C07312=1171.971,266.209,-67.189,-177.179,7.557,148.617
C07313=1171.975,265.960,-67.160,-177.181,7.554,148.617
C07314=1171.979,265.712,-67.133,-177.184,7.552,148.617
C07315=1171.984,265.463,-67.104,-177.186,7.549,148.617
C07316=1171.988,265.215,-67.077,-177.189,7.546,148.617
C07317=1171.992,264.966,-67.049,-177.192,7.543,148.617
C07318=1171.997,264.718,-67.020,-177.194,7.541,148.617
C07319=1172.002,264.470,-66.993,-177.197,7.538,148.617
C07320=1172.005,264.222,-66.964,-177.200,7.535,148.618
C07321=1172.011,263.973,-66.937,-177.202,7.532,148.618
C07322=1172.014,263.724,-66.909,-177.205,7.530,148.618
C07323=1172.019,263.476,-66.881,-177.208,7.527,148.618
C07324=1172.023,263.228,-66.853,-177.210,7.524,148.618
C07325=1172.028,262.979,-66.825,-177.213,7.521,148.618
C07326=1172.032,262.731,-66.797,-177.215,7.519,148.618
C07327=1172.037,262.458,-66.767,-177.219,7.515,148.618
C07328=1172.042,262.184,-66.736,-177.221,7.512,148.618
C07329=1172.047,261.912,-66.706,-177.224,7.509,148.618
C07330=1172.052,261.638,-66.675,-177.227,7.507,148.619
C07331=1172.055,261.390,-66.647,-177.230,7.504,148.619
C07332=1172.060,261.142,-66.619,-177.232,7.502,148.619
C07333=1172.064,260.894,-66.592,-177.235,7.499,148.619
C07334=1172.068,260.645,-66.564,-177.238,7.496,148.619
C07335=1172.073,260.396,-66.536,-177.241,7.493,148.619
C07336=1172.078,260.148,-66.508,-177.243,7.491,148.619
C07337=1172.082,259.900,-66.480,-177.245,7.488,148.619
C07338=1172.086,259.651,-66.453,-177.248,7.485,148.619
C07339=1172.091,259.403,-66.425,-177.251,7.482,148.619
C07340=1172.095,259.154,-66.398,-177.254,7.480,148.619
C07341=1172.099,258.906,-66.370,-177.256,7.477,148.619
C07342=1172.104,258.658,-66.343,-177.259,7.474,148.620
C07343=1172.107,258.409,-66.315,-177.261,7.472,148.620
C07344=1172.113,258.160,-66.287,-177.264,7.469,148.620
C07345=1172.117,257.913,-66.260,-177.267,7.466,148.620
C07346=1172.121,257.663,-66.232,-177.270,7.463,148.620
C07347=1172.126,257.415,-66.204,-177.272,7.461,148.620
C07348=1172.130,257.167,-66.177,-177.275,7.458,148.620
C07349=1172.135,256.919,-66.149,-177.278,7.455,148.620
C07350=1172.139,256.670,-66.122,-177.280,7.453,148.620
C07351=1172.143,256.421,-66.095,-177.283,7.450,148.620
C07352=1172.148,256.173,-66.067,-177.285,7.447,148.620
C07353=1172.152,255.924,-66.040,-177.288,7.444,148.620
C07354=1172.156,255.676,-66.013,-177.290,7.442,148.621
C07355=1172.161,255.428,-65.985,-177.294,7.439,148.621
C07356=1172.165,255.179,-65.958,-177.296,7.436,148.621
C07357=1172.170,254.931,-65.931,-177.298,7.434,148.621
C07358=1172.174,254.682,-65.903,-177.301,7.431,148.621
C07359=1172.178,254.434,-65.876,-177.304,7.428,148.621
C07360=1172.183,254.185,-65.849,-177.306,7.426,148.621
C07361=1172.187,253.937,-65.821,-177.309,7.424,148.622
C07362=1172.191,253.688,-65.793,-177.312,7.421,148.622
C07363=1172.196,253.440,-65.766,-177.315,7.418,148.622
C07364=1172.200,253.192,-65.740,-177.317,7.415,148.622
C07365=1172.204,252.944,-65.712,-177.320,7.413,148.622
C07366=1172.209,252.695,-65.685,-177.323,7.410,148.622
C07367=1172.213,252.446,-65.658,-177.325,7.408,148.622
C07368=1172.218,252.198,-65.631,-177.328,7.405,148.622
C07369=1172.222,251.949,-65.603,-177.331,7.402,148.622
C07370=1172.227,251.701,-65.576,-177.333,7.400,148.622
C07371=1172.231,251.453,-65.549,-177.336,7.397,148.622
C07372=1172.235,251.204,-65.522,-177.339,7.394,148.623
C07373=1172.239,250.955,-65.495,-177.341,7.392,148.623
C07374=1172.244,250.707,-65.468,-177.344,7.389,148.623
C07375=1172.249,250.458,-65.441,-177.346,7.386,148.623
C07376=1172.253,250.210,-65.414,-177.349,7.384,148.623
C07377=1172.258,249.961,-65.386,-177.352,7.381,148.623
C07378=1172.262,249.713,-65.360,-177.355,7.378,148.623
C07379=1172.266,249.464,-65.333,-177.357,7.376,148.623
C07380=1172.271,249.215,-65.306,-177.360,7.373,148.624
C07381=1172.275,248.967,-65.278,-177.363,7.371,148.624
C07382=1172.280,248.718,-65.251,-177.365,7.368,148.624
C07383=1172.284,248.470,-65.225,-177.368,7.365,148.624
C07384=1172.289,248.222,-65.198,-177.370,7.362,148.624
C07385=1172.293,247.973,-65.171,-177.373,7.360,148.624
C07386=1172.298,247.725,-65.144,-177.376,7.358,148.624
C07387=1172.302,247.477,-65.117,-177.379,7.355,148.624
C07388=1172.306,247.228,-65.090,-177.381,7.353,148.625
C07389=1172.310,246.979,-65.063,-177.384,7.350,148.625
C07390=1172.314,246.731,-65.036,-177.386,7.348,148.625
C07391=1172.319,246.482,-65.009,-177.389,7.345,148.625
C07392=1172.324,246.234,-64.982,-177.392,7.342,148.625
C07393=1172.328,245.985,-64.956,-177.394,7.340,148.625
C07394=1172.333,245.736,-64.929,-177.397,7.337,148.625
C07395=1172.337,245.488,-64.902,-177.400,7.334,148.626
C07396=1172.341,245.240,-64.876,-177.402,7.332,148.626
C07397=1172.346,244.991,-64.849,-177.405,7.329,148.626
C07398=1172.350,244.743,-64.822,-177.408,7.326,148.626
C07399=1172.355,244.494,-64.796,-177.410,7.324,148.626
C07400=1172.359,244.245,-64.769,-177.413,7.321,148.626
C07401=1172.364,243.997,-64.742,-177.416,7.320,148.627
C07402=1172.368,243.749,-64.715,-177.418,7.317,148.627
C07403=1172.373,243.500,-64.689,-177.421,7.314,148.627
C07404=1172.377,243.251,-64.663,-177.423,7.311,148.627
C07405=1172.381,243.003,-64.636,-177.427,7.309,148.627
C07406=1172.386,242.754,-64.610,-177.429,7.306,148.627
C07407=1172.390,242.506,-64.583,-177.431,7.304,148.627
C07408=1172.395,242.257,-64.556,-177.435,7.301,148.627
C07409=1172.399,242.008,-64.530,-177.437,7.299,148.628
C07410=1172.404,241.760,-64.503,-177.440,7.296,148.628
C07411=1172.408,241.512,-64.476,-177.443,7.293,148.628
C07412=1172.413,241.263,-64.450,-177.445,7.291,148.628
C07413=1172.417,241.014,-64.424,-177.448,7.288,148.628
C07414=1172.421,240.766,-64.396,-177.450,7.287,148.628
C07415=1172.426,240.517,-64.371,-177.453,7.284,148.629
C07416=1172.430,240.269,-64.344,-177.456,7.281,148.629
C07417=1172.434,240.020,-64.318,-177.458,7.278,148.629
C07418=1172.439,239.771,-64.291,-177.461,7.276,148.629
C07419=1172.443,239.522,-64.265,-177.464,7.274,148.629
C07420=1172.448,239.274,-64.238,-177.466,7.271,148.629
C07421=1172.453,239.026,-64.213,-177.469,7.268,148.629
C07422=1172.457,238.778,-64.186,-177.472,7.266,148.630
C07423=1172.462,238.529,-64.160,-177.474,7.263,148.630
C07424=1172.466,238.280,-64.133,-177.477,7.261,148.630
C07425=1172.471,238.031,-64.107,-177.480,7.258,148.630
C07426=1172.475,237.783,-64.081,-177.482,7.256,148.630
C07427=1172.479,237.534,-64.054,-177.485,7.253,148.630
C07428=1172.483,237.286,-64.028,-177.488,7.251,148.630
C07429=1172.488,237.037,-64.002,-177.491,7.249,148.631
C07430=1172.493,236.789,-63.976,-177.493,7.246,148.631
C07431=1172.498,236.517,-63.947,-177.496,7.243,148.631
C07432=1172.502,236.245,-63.919,-177.499,7.240,148.631
C07433=1172.507,235.974,-63.890,-177.502,7.238,148.631
C07434=1172.512,235.702,-63.862,-177.505,7.235,148.632
C07435=1172.516,235.454,-63.835,-177.508,7.232,148.632
C07436=1172.521,235.205,-63.809,-177.510,7.231,148.632
C07437=1172.525,234.956,-63.783,-177.513,7.228,148.632
C07438=1172.530,234.708,-63.757,-177.516,7.225,148.632
C07439=1172.535,234.459,-63.731,-177.518,7.223,148.632
C07440=1172.539,234.210,-63.705,-177.521,7.220,148.633
C07441=1172.543,233.962,-63.679,-177.524,7.218,148.633
C07442=1172.548,233.713,-63.652,-177.527,7.215,148.633
C07443=1172.553,233.465,-63.627,-177.529,7.213,148.633
C07444=1172.557,233.216,-63.601,-177.532,7.210,148.633
C07445=1172.561,232.967,-63.575,-177.534,7.208,148.633
C07446=1172.566,232.719,-63.548,-177.537,7.206,148.634
C07447=1172.570,232.470,-63.523,-177.540,7.204,148.634
C07448=1172.575,232.222,-63.497,-177.542,7.201,148.634
C07449=1172.579,231.973,-63.471,-177.546,7.198,148.634
C07450=1172.583,231.724,-63.446,-177.548,7.196,148.634
C07451=1172.588,231.475,-63.419,-177.551,7.193,148.635
C07452=1172.593,231.228,-63.393,-177.553,7.191,148.635
C07453=1172.597,230.979,-63.367,-177.556,7.188,148.635
C07454=1172.601,230.730,-63.342,-177.559,7.186,148.635
C07455=1172.605,230.481,-63.316,-177.561,7.183,148.635
C07456=1172.610,230.233,-63.291,-177.564,7.182,148.636
C07457=1172.615,229.984,-63.264,-177.567,7.179,148.636
C07458=1172.619,229.735,-63.239,-177.569,7.177,148.636
C07459=1172.624,229.487,-63.213,-177.572,7.174,148.636
C07460=1172.628,229.238,-63.187,-177.574,7.172,148.636
C07461=1172.633,228.990,-63.162,-177.578,7.169,148.636
C07462=1172.637,228.741,-63.136,-177.580,7.167,148.637
C07463=1172.642,228.493,-63.110,-177.583,7.164,148.637
C07464=1172.646,228.244,-63.085,-177.585,7.162,148.637
C07465=1172.650,227.995,-63.059,-177.588,7.160,148.637
C07466=1172.655,227.746,-63.033,-177.591,7.157,148.637
C07467=1172.660,227.498,-63.007,-177.594,7.155,148.638
C07468=1172.664,227.249,-62.982,-177.596,7.153,148.638
C07469=1172.668,227.000,-62.956,-177.599,7.150,148.638
C07470=1172.673,226.752,-62.930,-177.601,7.148,148.638
C07471=1172.678,226.503,-62.905,-177.604,7.145,148.638
C07472=1172.682,226.254,-62.880,-177.607,7.143,148.639
C07473=1172.687,226.006,-62.854,-177.610,7.140,148.639
C07474=1172.691,225.757,-62.828,-177.612,7.138,148.639
C07475=1172.696,225.509,-62.803,-177.615,7.136,148.639
C07476=1172.700,225.260,-62.777,-177.618,7.134,148.639
C07477=1172.704,225.011,-62.752,-177.620,7.131,148.640
C07478=1172.709,224.763,-62.727,-177.623,7.129,148.640
C07479=1172.714,224.514,-62.701,-177.626,7.126,148.640
C07480=1172.718,224.265,-62.675,-177.628,7.124,148.640
C07481=1172.723,224.017,-62.650,-177.631,7.121,148.640
C07482=1172.727,223.767,-62.625,-177.634,7.119,148.641
C07483=1172.732,223.519,-62.600,-177.637,7.117,148.641
C07484=1172.736,223.271,-62.574,-177.639,7.115,148.641
C07485=1172.740,223.022,-62.549,-177.642,7.112,148.641
C07486=1172.745,222.773,-62.524,-177.645,7.110,148.642
C07487=1172.749,222.525,-62.498,-177.647,7.108,148.642
C07488=1172.754,222.276,-62.473,-177.650,7.105,148.642
C07489=1172.758,222.027,-62.448,-177.652,7.103,148.642
C07490=1172.763,221.779,-62.422,-177.656,7.100,148.642
C07491=1172.768,221.530,-62.397,-177.658,7.098,148.642
C07492=1172.772,221.281,-62.372,-177.661,7.096,148.643
C07493=1172.777,221.033,-62.346,-177.663,7.094,148.643
C07494=1172.781,220.783,-62.322,-177.666,7.091,148.643
C07495=1172.786,220.535,-62.296,-177.669,7.089,148.643
C07496=1172.790,220.287,-62.271,-177.672,7.086,148.644
C07497=1172.795,220.038,-62.246,-177.674,7.084,148.644
C07498=1172.799,219.789,-62.220,-177.677,7.082,148.644
C07499=1172.803,219.541,-62.196,-177.679,7.079,148.644
C07500=1172.808,219.292,-62.170,-177.682,7.078,148.644
C07501=1172.813,219.043,-62.146,-177.685,7.075,148.645
C07502=1172.817,218.794,-62.120,-177.688,7.073,148.645
C07503=1172.822,218.546,-62.095,-177.690,7.070,148.645
C07504=1172.826,218.297,-62.070,-177.693,7.068,148.645
C07505=1172.831,218.048,-62.046,-177.696,7.065,148.646
C07506=1172.835,217.800,-62.020,-177.698,7.063,148.646
C07507=1172.840,217.551,-61.995,-177.701,7.062,148.646
C07508=1172.844,217.302,-61.970,-177.704,7.059,148.646
C07509=1172.849,217.054,-61.945,-177.706,7.057,148.646
C07510=1172.853,216.804,-61.920,-177.709,7.054,148.647
C07511=1172.857,216.556,-61.895,-177.712,7.052,148.647
C07512=1172.862,216.307,-61.870,-177.714,7.050,148.647
C07513=1172.867,216.059,-61.845,-177.717,7.047,148.647
C07514=1172.871,215.809,-61.820,-177.720,7.046,148.648
C07515=1172.876,215.561,-61.796,-177.723,7.043,148.648
C07516=1172.880,215.312,-61.770,-177.725,7.041,148.648
C07517=1172.885,215.063,-61.746,-177.728,7.038,148.648
C07518=1172.889,214.815,-61.721,-177.731,7.036,148.649
C07519=1172.894,214.566,-61.696,-177.733,7.034,148.649
C07520=1172.898,214.318,-61.672,-177.736,7.031,148.649
C07521=1172.903,214.068,-61.647,-177.739,7.030,148.649
C07522=1172.908,213.820,-61.622,-177.742,7.027,148.649
C07523=1172.911,213.571,-61.597,-177.744,7.025,148.650
C07524=1172.916,213.322,-61.572,-177.747,7.023,148.650
C07525=1172.921,213.074,-61.547,-177.750,7.020,148.650
C07526=1172.925,212.825,-61.523,-177.752,7.018,148.650
C07527=1172.930,212.577,-61.498,-177.755,7.015,148.651
C07528=1172.934,212.328,-61.474,-177.758,7.014,148.651
C07529=1172.939,212.079,-61.448,-177.760,7.011,148.651
C07530=1172.943,211.830,-61.424,-177.763,7.009,148.651
C07531=1172.948,211.581,-61.399,-177.765,7.007,148.651
C07532=1172.953,211.332,-61.375,-177.768,7.005,148.652
C07533=1172.957,211.084,-61.350,-177.771,7.002,148.652
C07534=1172.962,210.835,-61.325,-177.774,7.000,148.652
C07535=1172.967,210.565,-61.298,-177.777,6.998,148.653
C07536=1172.972,210.294,-61.273,-177.780,6.995,148.653
C07537=1172.976,210.023,-61.246,-177.782,6.993,148.653
C07538=1172.981,209.753,-61.219,-177.785,6.990,148.653
C07539=1172.986,209.505,-61.194,-177.788,6.988,148.654
C07540=1172.990,209.255,-61.170,-177.791,6.985,148.654
C07541=1172.995,209.007,-61.145,-177.794,6.984,148.654
C07542=1173.000,208.758,-61.121,-177.796,6.982,148.654
C07543=1173.005,208.510,-61.096,-177.799,6.979,148.655
C07544=1173.009,208.260,-61.072,-177.802,6.977,148.655
C07545=1173.014,208.012,-61.047,-177.804,6.975,148.655
C07546=1173.018,207.763,-61.023,-177.807,6.972,148.655
C07547=1173.022,207.514,-60.999,-177.810,6.971,148.656
C07548=1173.027,207.265,-60.974,-177.813,6.968,148.656
C07549=1173.031,207.017,-60.950,-177.815,6.966,148.656
C07550=1173.037,206.768,-60.925,-177.818,6.964,148.656
C07551=1173.040,206.519,-60.901,-177.821,6.961,148.657
C07552=1173.045,206.271,-60.877,-177.823,6.959,148.657
C07553=1173.050,206.022,-60.852,-177.826,6.958,148.657
C07554=1173.054,205.774,-60.828,-177.829,6.955,148.657
C07555=1173.059,205.524,-60.804,-177.831,6.953,148.658
C07556=1173.064,205.275,-60.780,-177.834,6.951,148.658
C07557=1173.068,205.027,-60.756,-177.837,6.948,148.658
C07558=1173.073,204.778,-60.731,-177.839,6.946,148.658
C07559=1173.077,204.529,-60.707,-177.842,6.945,148.659
C07560=1173.081,204.281,-60.683,-177.845,6.942,148.659
C07561=1173.087,204.031,-60.659,-177.848,6.940,148.659
C07562=1173.091,203.783,-60.634,-177.850,6.938,148.659
C07563=1173.096,203.534,-60.610,-177.853,6.935,148.660
C07564=1173.099,203.285,-60.586,-177.856,6.933,148.660
C07565=1173.105,203.036,-60.562,-177.858,6.931,148.660
C07566=1173.109,202.788,-60.538,-177.861,6.929,148.660
C07567=1173.114,202.539,-60.514,-177.864,6.927,148.661
C07568=1173.118,202.291,-60.490,-177.866,6.925,148.661
C07569=1173.123,202.041,-60.465,-177.869,6.922,148.661
C07570=1173.127,201.792,-60.441,-177.872,6.920,148.662
C07571=1173.132,201.544,-60.417,-177.875,6.918,148.662
C07572=1173.136,201.295,-60.394,-177.877,6.916,148.662
C07573=1173.141,201.046,-60.369,-177.880,6.914,148.662
C07574=1173.146,200.798,-60.345,-177.883,6.912,148.663
C07575=1173.150,200.548,-60.321,-177.885,6.910,148.663
C07576=1173.154,200.299,-60.297,-177.888,6.907,148.663
C07577=1173.159,200.050,-60.274,-177.891,6.905,148.664
C07578=1173.164,199.802,-60.249,-177.893,6.903,148.664
C07579=1173.168,199.553,-60.225,-177.896,6.901,148.664
C07580=1173.173,199.304,-60.202,-177.899,6.899,148.664
C07581=1173.178,199.056,-60.178,-177.901,6.897,148.664
C07582=1173.182,198.807,-60.155,-177.904,6.894,148.665
C07583=1173.187,198.558,-60.130,-177.907,6.892,148.665
C07584=1173.191,198.309,-60.107,-177.910,6.891,148.665
C07585=1173.196,198.060,-60.082,-177.912,6.889,148.666
C07586=1173.201,197.811,-60.059,-177.915,6.886,148.666
C07587=1173.205,197.563,-60.035,-177.918,6.884,148.666
C07588=1173.210,197.313,-60.011,-177.920,6.882,148.666
C07589=1173.214,197.065,-59.987,-177.923,6.879,148.667
C07590=1173.219,196.816,-59.964,-177.926,6.878,148.667
C07591=1173.223,196.568,-59.940,-177.929,6.876,148.667
C07592=1173.228,196.319,-59.916,-177.931,6.874,148.668
C07593=1173.233,196.070,-59.893,-177.934,6.871,148.668
C07594=1173.237,195.821,-59.869,-177.937,6.869,148.668
C07595=1173.242,195.572,-59.846,-177.939,6.867,148.668
C07596=1173.246,195.324,-59.822,-177.942,6.865,148.669
C07597=1173.251,195.075,-59.798,-177.945,6.863,148.669
C07598=1173.255,194.826,-59.775,-177.947,6.861,148.669
C07599=1173.260,194.577,-59.751,-177.950,6.859,148.670
C07600=1173.264,194.328,-59.727,-177.953,6.856,148.670
C07601=1173.269,194.078,-59.704,-177.956,6.855,148.670
C07602=1173.273,193.830,-59.680,-177.958,6.853,148.671
C07603=1173.278,193.581,-59.656,-177.960,6.851,148.671
C07604=1173.282,193.332,-59.633,-177.964,6.848,148.671
C07605=1173.287,193.083,-59.610,-177.966,6.846,148.671
C07606=1173.292,192.835,-59.585,-177.969,6.845,148.672
C07607=1173.297,192.586,-59.562,-177.971,6.842,148.672
C07608=1173.302,192.337,-59.539,-177.974,6.840,148.672
C07609=1173.306,192.088,-59.516,-177.977,6.838,148.673
C07610=1173.311,191.840,-59.492,-177.980,6.836,148.673
C07611=1173.315,191.591,-59.468,-177.982,6.834,148.673
C07612=1173.320,191.342,-59.445,-177.985,6.832,148.673
C07613=1173.325,191.093,-59.422,-177.988,6.830,148.674
C07614=1173.329,190.844,-59.398,-177.991,6.828,148.674
C07615=1173.334,190.595,-59.374,-177.993,6.826,148.674
C07616=1173.338,190.346,-59.351,-177.996,6.824,148.675
C07617=1173.343,190.097,-59.328,-177.999,6.822,148.675
C07618=1173.347,189.848,-59.305,-178.001,6.820,148.675
C07619=1173.352,189.599,-59.281,-178.004,6.818,148.675
C07620=1173.357,189.350,-59.258,-178.006,6.816,148.676
C07621=1173.361,189.101,-59.235,-178.010,6.813,148.676
C07622=1173.366,188.852,-59.211,-178.012,6.811,148.676
C07623=1173.370,188.604,-59.188,-178.014,6.809,148.677
C07624=1173.375,188.355,-59.165,-178.017,6.808,148.677
C07625=1173.380,188.106,-59.142,-178.020,6.805,148.677
C07626=1173.385,187.857,-59.119,-178.023,6.803,148.678
C07627=1173.389,187.608,-59.095,-178.026,6.801,148.678
C07628=1173.393,187.359,-59.073,-178.028,6.799,148.678
C07629=1173.398,187.110,-59.049,-178.031,6.798,148.678
C07630=1173.403,186.861,-59.026,-178.034,6.795,148.679
C07631=1173.407,186.612,-59.003,-178.037,6.793,148.679
C07632=1173.412,186.364,-58.980,-178.039,6.791,148.679
C07633=1173.417,186.115,-58.957,-178.041,6.789,148.680
C07634=1173.421,185.866,-58.933,-178.044,6.787,148.680
C07635=1173.426,185.617,-58.910,-178.047,6.785,148.680
C07636=1173.430,185.368,-58.887,-178.050,6.783,148.681
C07637=1173.435,185.119,-58.864,-178.053,6.781,148.681
C07638=1173.439,184.870,-58.841,-178.055,6.779,148.681
C07639=1173.444,184.601,-58.816,-178.058,6.777,148.681
C07640=1173.449,184.331,-58.791,-178.061,6.775,148.682
C07641=1173.455,184.061,-58.766,-178.064,6.772,148.682
C07642=1173.459,183.792,-58.742,-178.067,6.771,148.682
C07643=1173.465,183.544,-58.719,-178.069,6.769,148.683
C07644=1173.469,183.295,-58.695,-178.072,6.767,148.683
C07645=1173.473,183.046,-58.673,-178.075,6.764,148.684
C07646=1173.478,182.797,-58.649,-178.078,6.763,148.684
C07647=1173.483,182.547,-58.627,-178.080,6.760,148.684
C07648=1173.487,182.299,-58.604,-178.083,6.759,148.684
C07649=1173.492,182.050,-58.581,-178.086,6.757,148.685
C07650=1173.496,181.801,-58.558,-178.088,6.755,148.685
C07651=1173.501,181.552,-58.535,-178.091,6.753,148.685
C07652=1173.506,181.303,-58.512,-178.094,6.751,148.686
C07653=1173.510,181.055,-58.490,-178.096,6.749,148.686
C07654=1173.515,180.806,-58.466,-178.099,6.747,148.686
C07655=1173.519,180.556,-58.444,-178.102,6.745,148.687
C07656=1173.524,180.307,-58.421,-178.104,6.743,148.687
C07657=1173.529,180.059,-58.398,-178.108,6.741,148.687
C07658=1173.534,179.810,-58.376,-178.110,6.739,148.688
C07659=1173.538,179.561,-58.352,-178.113,6.737,148.688
C07660=1173.542,179.312,-58.330,-178.115,6.735,148.688
C07661=1173.548,179.063,-58.307,-178.118,6.733,148.689
C07662=1173.552,178.814,-58.285,-178.121,6.732,148.689
C07663=1173.557,178.565,-58.262,-178.124,6.729,148.689
C07664=1173.561,178.317,-58.240,-178.127,6.727,148.690
C07665=1173.566,178.068,-58.216,-178.129,6.725,148.690
C07666=1173.570,177.818,-58.194,-178.131,6.723,148.690
C07667=1173.576,177.570,-58.171,-178.134,6.722,148.691
C07668=1173.580,177.321,-58.149,-178.137,6.720,148.691
C07669=1173.585,177.071,-58.126,-178.139,6.718,148.691
C07670=1173.589,176.822,-58.104,-178.143,6.715,148.692
C07671=1173.594,176.574,-58.081,-178.145,6.714,148.692
C07672=1173.599,176.324,-58.059,-178.148,6.712,148.692
C07673=1173.602,176.076,-58.036,-178.151,6.710,148.693
C07674=1173.608,175.827,-58.014,-178.153,6.708,148.693
C07675=1173.612,175.578,-57.991,-178.156,6.706,148.693
C07676=1173.617,175.328,-57.968,-178.158,6.704,148.694
C07677=1173.622,175.080,-57.946,-178.161,6.703,148.694
C07678=1173.626,174.831,-57.924,-178.164,6.700,148.694
C07679=1173.631,174.582,-57.902,-178.167,6.698,148.695
C07680=1173.635,174.333,-57.879,-178.170,6.697,148.695
C07681=1173.640,174.084,-57.856,-178.172,6.695,148.695
C07682=1173.645,173.836,-57.834,-178.174,6.693,148.695
C07683=1173.649,173.586,-57.812,-178.177,6.691,148.696
C07684=1173.654,173.337,-57.789,-178.180,6.689,148.696
C07685=1173.659,173.089,-57.767,-178.183,6.687,148.697
C07686=1173.663,172.839,-57.745,-178.186,6.685,148.697
C07687=1173.669,172.590,-57.722,-178.188,6.683,148.697
C07688=1173.673,172.342,-57.700,-178.191,6.681,148.698
C07689=1173.678,172.093,-57.678,-178.194,6.680,148.698
C07690=1173.683,171.843,-57.655,-178.197,6.678,148.698
C07691=1173.687,171.595,-57.632,-178.199,6.676,148.699
C07692=1173.691,171.346,-57.611,-178.201,6.674,148.699
C07693=1173.696,171.097,-57.589,-178.204,6.672,148.699
C07694=1173.701,170.848,-57.566,-178.207,6.670,148.700
C07695=1173.705,170.599,-57.544,-178.209,6.669,148.700
C07696=1173.710,170.350,-57.522,-178.213,6.666,148.700
C07697=1173.715,170.101,-57.499,-178.215,6.664,148.701
C07698=1173.719,169.851,-57.477,-178.218,6.662,148.701
C07699=1173.724,169.603,-57.456,-178.221,6.661,148.701
C07700=1173.728,169.354,-57.433,-178.223,6.659,148.702
C07701=1173.733,169.105,-57.411,-178.226,6.657,148.702
C07702=1173.738,168.856,-57.389,-178.229,6.655,148.703
C07703=1173.743,168.607,-57.367,-178.232,6.654,148.703
C07704=1173.747,168.358,-57.345,-178.234,6.652,148.703
C07705=1173.752,168.109,-57.323,-178.236,6.650,148.703
C07706=1173.757,167.859,-57.300,-178.239,6.648,148.704
C07707=1173.762,167.611,-57.279,-178.242,6.646,148.704
C07708=1173.766,167.362,-57.256,-178.244,6.645,148.705
C07709=1173.771,167.113,-57.234,-178.248,6.642,148.705
C07710=1173.775,166.864,-57.212,-178.250,6.640,148.705
C07711=1173.780,166.615,-57.191,-178.253,6.638,148.706
C07712=1173.784,166.366,-57.169,-178.256,6.637,148.706
C07713=1173.790,166.117,-57.146,-178.258,6.635,148.706
C07714=1173.795,165.869,-57.125,-178.261,6.633,148.707
C07715=1173.799,165.619,-57.103,-178.264,6.631,148.707
C07716=1173.804,165.371,-57.081,-178.267,6.630,148.707
C07717=1173.808,165.121,-57.059,-178.269,6.628,148.708
C07718=1173.813,164.873,-57.037,-178.272,6.626,148.708
C07719=1173.817,164.623,-57.015,-178.275,6.624,148.709
C07720=1173.822,164.375,-56.993,-178.277,6.623,148.709
C07721=1173.826,164.125,-56.971,-178.280,6.621,148.709
C07722=1173.831,163.877,-56.950,-178.283,6.619,148.710
C07723=1173.836,163.627,-56.928,-178.285,6.617,148.710
C07724=1173.841,163.378,-56.907,-178.288,6.616,148.710
C07725=1173.846,163.129,-56.884,-178.291,6.614,148.711
C07726=1173.851,162.880,-56.862,-178.293,6.612,148.711
C07727=1173.855,162.631,-56.841,-178.296,6.610,148.711
C07728=1173.860,162.382,-56.819,-178.299,6.607,148.712
C07729=1173.865,162.133,-56.797,-178.302,6.606,148.712
C07730=1173.869,161.884,-56.775,-178.304,6.604,148.712
C07731=1173.874,161.634,-56.754,-178.307,6.602,148.713
C07732=1173.879,161.386,-56.732,-178.310,6.600,148.713
C07733=1173.884,161.137,-56.711,-178.312,6.598,148.714
C07734=1173.887,160.888,-56.689,-178.315,6.597,148.714
C07735=1173.892,160.640,-56.667,-178.318,6.595,148.714
C07736=1173.897,160.390,-56.646,-178.320,6.593,148.715
C07737=1173.902,160.141,-56.624,-178.323,6.591,148.715
C07738=1173.906,159.892,-56.603,-178.326,6.590,148.715
C07739=1173.911,159.643,-56.581,-178.328,6.588,148.716
C07740=1173.916,159.394,-56.560,-178.331,6.586,148.716
C07741=1173.921,159.145,-56.538,-178.334,6.584,148.717
C07742=1173.925,158.896,-56.516,-178.336,6.583,148.717
C07743=1173.931,158.626,-56.493,-178.339,6.581,148.717
C07744=1173.935,158.357,-56.470,-178.342,6.580,148.718
C07745=1173.940,158.090,-56.447,-178.346,6.577,148.718
C07746=1173.946,157.820,-56.423,-178.348,6.575,148.719
C07747=1173.950,157.571,-56.401,-178.351,6.573,148.719
C07748=1173.955,157.322,-56.380,-178.354,6.572,148.719
C07749=1173.960,157.073,-56.359,-178.356,6.570,148.720
C07750=1173.964,156.824,-56.337,-178.359,6.568,148.720
C07751=1173.969,156.575,-56.316,-178.362,6.566,148.720
C07752=1173.974,156.326,-56.295,-178.364,6.565,148.721
C07753=1173.979,156.077,-56.274,-178.367,6.563,148.721
C07754=1173.983,155.827,-56.252,-178.370,6.561,148.722
C07755=1173.988,155.578,-56.231,-178.373,6.559,148.722
C07756=1173.992,155.330,-56.210,-178.375,6.558,148.722
C07757=1173.997,155.081,-56.188,-178.378,6.556,148.723
C07758=1174.002,154.831,-56.166,-178.381,6.554,148.723
C07759=1174.007,154.583,-56.145,-178.383,6.552,148.723
C07760=1174.012,154.333,-56.124,-178.386,6.551,148.724
C07761=1174.016,154.085,-56.103,-178.389,6.549,148.724
C07762=1174.021,153.835,-56.081,-178.391,6.547,148.725
C07763=1174.025,153.586,-56.060,-178.394,6.545,148.725
C07764=1174.031,153.337,-56.039,-178.397,6.544,148.725
C07765=1174.035,153.088,-56.018,-178.399,6.542,148.726
C07766=1174.039,152.839,-55.996,-178.402,6.540,148.726
C07767=1174.045,152.590,-55.975,-178.404,6.539,148.727
C07768=1174.049,152.341,-55.954,-178.407,6.538,148.727
C07769=1174.054,152.092,-55.933,-178.410,6.536,148.728
C07770=1174.059,151.843,-55.912,-178.413,6.534,148.728
C07771=1174.063,151.593,-55.890,-178.415,6.532,148.728
C07772=1174.068,151.344,-55.870,-178.418,6.531,148.729
C07773=1174.073,151.096,-55.848,-178.421,6.529,148.729
C07774=1174.078,150.847,-55.827,-178.424,6.527,148.729
C07775=1174.082,150.598,-55.807,-178.426,6.525,148.730
C07776=1174.087,150.349,-55.785,-178.429,6.524,148.730
C07777=1174.092,150.099,-55.764,-178.432,6.522,148.731
C07778=1174.096,149.850,-55.744,-178.434,6.520,148.731
C07779=1174.101,149.601,-55.722,-178.437,6.518,148.731
C07780=1174.106,149.352,-55.701,-178.440,6.517,148.732
C07781=1174.111,149.103,-55.681,-178.442,6.515,148.732
C07782=1174.116,148.854,-55.660,-178.445,6.513,148.732
C07783=1174.120,148.606,-55.638,-178.448,6.511,148.733
C07784=1174.124,148.356,-55.617,-178.450,6.510,148.733
C07785=1174.130,148.106,-55.596,-178.454,6.508,148.734
C07786=1174.134,147.857,-55.576,-178.456,6.507,148.734
C07787=1174.139,147.609,-55.554,-178.458,6.506,148.735
C07788=1174.143,147.360,-55.534,-178.461,6.504,148.735
C07789=1174.149,147.111,-55.513,-178.464,6.502,148.735
C07790=1174.153,146.862,-55.492,-178.467,6.500,148.736
C07791=1174.158,146.612,-55.471,-178.469,6.499,148.736
C07792=1174.163,146.363,-55.450,-178.472,6.497,148.736
C07793=1174.167,146.114,-55.429,-178.475,6.495,148.737
C07794=1174.172,145.865,-55.408,-178.477,6.493,148.737
C07795=1174.176,145.616,-55.388,-178.480,6.492,148.738
C07796=1174.182,145.367,-55.367,-178.483,6.490,148.738
C07797=1174.186,145.118,-55.346,-178.486,6.488,148.739
C07798=1174.191,144.868,-55.325,-178.489,6.487,148.739
C07799=1174.196,144.620,-55.305,-178.491,6.486,148.739
C07800=1174.201,144.370,-55.284,-178.493,6.484,148.740
C07801=1174.205,144.121,-55.264,-178.496,6.482,148.740
C07802=1174.210,143.872,-55.243,-178.499,6.481,148.741
C07803=1174.215,143.623,-55.222,-178.501,6.479,148.741
C07804=1174.219,143.374,-55.202,-178.504,6.477,148.741
C07805=1174.224,143.126,-55.180,-178.507,6.475,148.742
C07806=1174.229,142.877,-55.160,-178.510,6.474,148.742
C07807=1174.234,142.627,-55.139,-178.513,6.472,148.743
C07808=1174.239,142.378,-55.119,-178.515,6.470,148.743
C07809=1174.244,142.128,-55.098,-178.518,6.469,148.744
C07810=1174.248,141.880,-55.078,-178.520,6.468,148.744
C07811=1174.253,141.631,-55.058,-178.523,6.466,148.744
C07812=1174.258,141.381,-55.037,-178.526,6.464,148.745
C07813=1174.262,141.132,-55.016,-178.528,6.462,148.745
C07814=1174.267,140.883,-54.996,-178.531,6.461,148.745
C07815=1174.272,140.634,-54.975,-178.534,6.459,148.746
C07816=1174.276,140.385,-54.955,-178.537,6.458,148.746
C07817=1174.281,140.136,-54.934,-178.540,6.456,148.747
C07818=1174.286,139.887,-54.913,-178.542,6.455,148.747
C07819=1174.290,139.638,-54.893,-178.544,6.453,148.748
C07820=1174.296,139.388,-54.873,-178.547,6.451,148.748
C07821=1174.300,139.139,-54.852,-178.550,6.450,148.748
C07822=1174.305,138.890,-54.832,-178.553,6.448,148.749
C07823=1174.309,138.641,-54.811,-178.556,6.447,148.749
C07824=1174.314,138.392,-54.790,-178.558,6.445,148.750
C07825=1174.319,138.143,-54.770,-178.561,6.443,148.750
C07826=1174.323,137.894,-54.750,-178.563,6.442,148.751
C07827=1174.329,137.644,-54.729,-178.566,6.440,148.751
C07828=1174.333,137.395,-54.709,-178.569,6.439,148.751
C07829=1174.338,137.146,-54.689,-178.571,6.437,148.752
C07830=1174.342,136.897,-54.669,-178.575,6.436,148.752
C07831=1174.347,136.648,-54.648,-178.577,6.434,148.753
C07832=1174.352,136.399,-54.628,-178.580,6.432,148.753
C07833=1174.357,136.150,-54.608,-178.582,6.431,148.754
C07834=1174.362,135.901,-54.588,-178.585,6.429,148.754
C07835=1174.367,135.652,-54.567,-178.587,6.428,148.754
C07836=1174.371,135.403,-54.547,-178.590,6.426,148.755
C07837=1174.376,135.153,-54.527,-178.593,6.424,148.755
C07838=1174.380,134.904,-54.507,-178.596,6.423,148.756
C07839=1174.385,134.655,-54.486,-178.598,6.422,148.756
C07840=1174.390,134.405,-54.466,-178.601,6.420,148.756
C07841=1174.395,134.157,-54.446,-178.604,6.418,148.757
C07842=1174.400,133.908,-54.426,-178.606,6.417,148.757
C07843=1174.405,133.658,-54.406,-178.609,6.415,148.758
C07844=1174.409,133.410,-54.386,-178.612,6.413,148.758
C07845=1174.415,133.160,-54.365,-178.615,6.412,148.759
C07846=1174.419,132.911,-54.345,-178.617,6.411,148.759
C07847=1174.424,132.642,-54.324,-178.620,6.409,148.759
C07848=1174.429,132.374,-54.302,-178.623,6.408,148.760
C07849=1174.434,132.105,-54.280,-178.626,6.406,148.760
C07850=1174.440,131.836,-54.259,-178.629,6.403,148.761
C07851=1174.444,131.587,-54.238,-178.631,6.403,148.761
C07852=1174.450,131.338,-54.219,-178.634,6.401,148.762
C07853=1174.454,131.089,-54.199,-178.637,6.399,148.762
C07854=1174.459,130.840,-54.179,-178.640,6.398,148.763
C07855=1174.463,130.591,-54.159,-178.642,6.396,148.763
C07856=1174.468,130.341,-54.139,-178.645,6.395,148.764
C07857=1174.473,130.093,-54.119,-178.648,6.394,148.764
C07858=1174.478,129.843,-54.099,-178.650,6.392,148.764
C07859=1174.482,129.594,-54.079,-178.653,6.390,148.765
C07860=1174.487,129.345,-54.059,-178.656,6.388,148.765
C07861=1174.492,129.096,-54.040,-178.658,6.387,148.766
C07862=1174.497,128.847,-54.020,-178.661,6.386,148.766
C07863=1174.501,128.598,-54.000,-178.664,6.384,148.767
C07864=1174.506,128.349,-53.980,-178.666,6.383,148.767
C07865=1174.511,128.100,-53.960,-178.669,6.381,148.767
C07866=1174.516,127.850,-53.941,-178.671,6.380,148.768
C07867=1174.520,127.601,-53.920,-178.674,6.378,148.768
C07868=1174.525,127.352,-53.901,-178.677,6.377,148.769
C07869=1174.530,127.103,-53.881,-178.680,6.375,148.769
C07870=1174.535,126.854,-53.861,-178.682,6.373,148.770
C07871=1174.540,126.604,-53.841,-178.685,6.373,148.770
C07872=1174.544,126.355,-53.822,-178.688,6.371,148.771
C07873=1174.549,126.106,-53.802,-178.691,6.369,148.771
C07874=1174.554,125.857,-53.782,-178.693,6.367,148.771
C07875=1174.559,125.607,-53.762,-178.695,6.367,148.772
C07876=1174.564,125.358,-53.743,-178.699,6.365,148.772
C07877=1174.569,125.109,-53.723,-178.701,6.363,148.773
C07878=1174.573,124.860,-53.703,-178.704,6.362,148.773
C07879=1174.578,124.610,-53.683,-178.707,6.360,148.774
C07880=1174.584,124.361,-53.664,-178.709,6.359,148.774
C07881=1174.587,124.113,-53.644,-178.712,6.358,148.775
C07882=1174.592,123.863,-53.625,-178.715,6.356,148.775
C07883=1174.597,123.614,-53.605,-178.717,6.354,148.775
C07884=1174.602,123.365,-53.586,-178.719,6.353,148.776
C07885=1174.607,123.115,-53.566,-178.723,6.352,148.777
C07886=1174.612,122.866,-53.547,-178.725,6.350,148.777
C07887=1174.617,122.617,-53.526,-178.728,6.348,148.777
C07888=1174.621,122.368,-53.507,-178.730,6.348,148.778
C07889=1174.626,122.119,-53.488,-178.733,6.346,148.778
C07890=1174.631,121.870,-53.468,-178.736,6.344,148.779
C07891=1174.635,121.620,-53.449,-178.739,6.343,148.779
C07892=1174.641,121.371,-53.430,-178.741,6.342,148.780
C07893=1174.645,121.122,-53.410,-178.744,6.340,148.780
C07894=1174.650,120.873,-53.391,-178.747,6.339,148.781
C07895=1174.655,120.624,-53.371,-178.750,6.337,148.781
C07896=1174.660,120.374,-53.352,-178.752,6.336,148.781
C07897=1174.665,120.125,-53.333,-178.754,6.334,148.782
C07898=1174.669,119.876,-53.313,-178.758,6.333,148.782
C07899=1174.674,119.627,-53.294,-178.760,6.331,148.783
C07900=1174.679,119.377,-53.275,-178.762,6.330,148.783
C07901=1174.684,119.128,-53.255,-178.766,6.329,148.784
C07902=1174.689,118.879,-53.236,-178.768,6.327,148.784
C07903=1174.693,118.630,-53.217,-178.771,6.325,148.785
C07904=1174.698,118.381,-53.197,-178.773,6.324,148.785
C07905=1174.703,118.131,-53.178,-178.776,6.323,148.786
C07906=1174.707,117.882,-53.159,-178.779,6.321,148.786
C07907=1174.713,117.633,-53.139,-178.782,6.320,148.786
C07908=1174.717,117.384,-53.120,-178.784,6.319,148.787
C07909=1174.723,117.135,-53.100,-178.787,6.317,148.788
C07910=1174.727,116.886,-53.081,-178.790,6.316,148.788
C07911=1174.732,116.637,-53.062,-178.792,6.315,148.788
C07912=1174.737,116.387,-53.042,-178.795,6.313,148.789
C07913=1174.741,116.139,-53.024,-178.798,6.312,148.789
C07914=1174.746,115.888,-53.005,-178.801,6.310,148.790
C07915=1174.752,115.640,-52.985,-178.803,6.309,148.790
C07916=1174.756,115.390,-52.966,-178.805,6.307,148.791
C07917=1174.761,115.141,-52.947,-178.809,6.306,148.791
C07918=1174.765,114.892,-52.928,-178.811,6.305,148.792
C07919=1174.770,114.643,-52.909,-178.813,6.303,148.792
C07920=1174.775,114.393,-52.890,-178.817,6.302,148.793
C07921=1174.780,114.145,-52.871,-178.819,6.301,148.793
C07922=1174.785,113.895,-52.851,-178.821,6.299,148.793
C07923=1174.790,113.646,-52.832,-178.824,6.297,148.794
C07924=1174.794,113.397,-52.813,-178.827,6.296,148.794
C07925=1174.800,113.147,-52.794,-178.829,6.295,148.795
C07926=1174.804,112.898,-52.775,-178.832,6.293,148.795
C07927=1174.809,112.649,-52.756,-178.835,6.292,148.796
C07928=1174.813,112.399,-52.738,-178.837,6.291,148.796
C07929=1174.819,112.150,-52.718,-178.840,6.289,148.797
C07930=1174.824,111.901,-52.699,-178.843,6.288,148.797
C07931=1174.828,111.652,-52.680,-178.846,6.287,148.798
C07932=1174.833,111.402,-52.661,-178.848,6.285,148.798
C07933=1174.838,111.154,-52.642,-178.851,6.284,148.799
C07934=1174.843,110.905,-52.623,-178.854,6.283,148.799
C07935=1174.847,110.655,-52.605,-178.856,6.281,148.800
C07936=1174.853,110.406,-52.586,-178.859,6.280,148.800
C07937=1174.857,110.156,-52.567,-178.862,6.279,148.801
C07938=1174.862,109.907,-52.548,-178.864,6.277,148.801
C07939=1174.866,109.658,-52.529,-178.867,6.276,148.801
C07940=1174.872,109.408,-52.510,-178.870,6.275,148.802
C07941=1174.877,109.160,-52.492,-178.872,6.273,148.803
C07942=1174.882,108.910,-52.473,-178.875,6.272,148.803
C07943=1174.886,108.661,-52.454,-178.877,6.271,148.803
C07944=1174.890,108.412,-52.435,-178.880,6.269,148.804
C07945=1174.896,108.162,-52.416,-178.883,6.268,148.804
C07946=1174.901,107.914,-52.398,-178.885,6.267,148.805
C07947=1174.906,107.664,-52.379,-178.888,6.265,148.805
C07948=1174.910,107.415,-52.360,-178.891,6.264,148.806
C07949=1174.916,107.166,-52.341,-178.893,6.263,148.806
C07950=1174.920,106.916,-52.322,-178.896,6.261,148.807
C07951=1174.925,106.648,-52.303,-178.899,6.260,148.807
C07952=1174.931,106.380,-52.283,-178.902,6.258,148.808
C07953=1174.936,106.111,-52.262,-178.905,6.257,148.808
C07954=1174.941,105.843,-52.242,-178.908,6.256,148.809
C07955=1174.946,105.594,-52.223,-178.910,6.254,148.809
C07956=1174.951,105.344,-52.205,-178.913,6.253,148.810
C07957=1174.955,105.095,-52.187,-178.916,6.252,148.810
C07958=1174.961,104.846,-52.168,-178.918,6.250,148.811
C07959=1174.965,104.596,-52.149,-178.921,6.249,148.811
C07960=1174.970,104.347,-52.130,-178.924,6.248,148.812
C07961=1174.975,104.098,-52.112,-178.927,6.246,148.812
C07962=1174.980,103.848,-52.094,-178.929,6.245,148.813
C07963=1174.984,103.600,-52.075,-178.932,6.244,148.813
C07964=1174.990,103.350,-52.056,-178.935,6.242,148.814
C07965=1174.994,103.100,-52.038,-178.937,6.241,148.814
C07966=1174.999,102.852,-52.019,-178.940,6.240,148.815
C07967=1175.004,102.602,-52.001,-178.943,6.238,148.815
C07968=1175.009,102.353,-51.983,-178.945,6.237,148.816
C07969=1175.013,102.104,-51.964,-178.948,6.236,148.816
C07970=1175.018,101.855,-51.946,-178.951,6.234,148.817
C07971=1175.023,101.605,-51.928,-178.953,6.233,148.817
C07972=1175.029,101.357,-51.908,-178.956,6.232,148.818
C07973=1175.033,101.107,-51.890,-178.958,6.231,148.818
C07974=1175.038,100.857,-51.872,-178.961,6.230,148.819
C07975=1175.043,100.608,-51.854,-178.964,6.228,148.819
C07976=1175.048,100.359,-51.835,-178.966,6.227,148.820
C07977=1175.052,100.110,-51.816,-178.969,6.226,148.820
C07978=1175.057,99.860,-51.798,-178.971,6.225,148.821
C07979=1175.062,99.611,-51.780,-178.974,6.223,148.821
C07980=1175.067,99.362,-51.762,-178.977,6.222,148.822
C07981=1175.072,99.112,-51.743,-178.980,6.221,148.822
C07982=1175.077,98.863,-51.725,-178.982,6.219,148.823
C07983=1175.082,98.614,-51.707,-178.985,6.219,148.823
C07984=1175.087,98.365,-51.689,-178.988,6.217,148.824
C07985=1175.091,98.115,-51.671,-178.990,6.215,148.824
C07986=1175.096,97.866,-51.653,-178.993,6.215,148.825
C07987=1175.101,97.616,-51.634,-178.996,6.213,148.825
C07988=1175.106,97.367,-51.616,-178.998,6.212,148.826
C07989=1175.111,97.119,-51.597,-179.001,6.211,148.826
C07990=1175.115,96.869,-51.579,-179.004,6.209,148.827
C07991=1175.120,96.620,-51.561,-179.006,6.209,148.827
C07992=1175.125,96.370,-51.543,-179.009,6.207,148.828
C07993=1175.130,96.121,-51.525,-179.011,6.206,148.828
C07994=1175.135,95.872,-51.507,-179.014,6.205,148.829
C07995=1175.141,95.623,-51.488,-179.017,6.204,148.829
C07996=1175.145,95.373,-51.470,-179.020,6.202,148.830
C07997=1175.150,95.124,-51.452,-179.022,6.201,148.830
C07998=1175.155,94.874,-51.434,-179.025,6.200,148.831
C07999=1175.160,94.625,-51.416,-179.028,6.198,148.831
C08000=1175.165,94.376,-51.398,-179.030,6.197,148.832
C08001=1175.169,94.127,-51.380,-179.033,6.196,148.832
C08002=1175.174,93.878,-51.362,-179.035,6.195,148.833
C08003=1175.179,93.628,-51.344,-179.038,6.193,148.833
C08004=1175.184,93.379,-51.326,-179.041,6.192,148.834
C08005=1175.188,93.129,-51.308,-179.043,6.191,148.834
C08006=1175.193,92.880,-51.290,-179.046,6.189,148.835
C08007=1175.198,92.631,-51.272,-179.049,6.189,148.835
C08008=1175.203,92.382,-51.254,-179.051,6.187,148.836
C08009=1175.208,92.132,-51.237,-179.054,6.187,148.836
C08010=1175.213,91.883,-51.219,-179.057,6.185,148.837
C08011=1175.218,91.634,-51.201,-179.059,6.184,148.837
C08012=1175.223,91.385,-51.183,-179.062,6.183,148.838
C08013=1175.227,91.135,-51.164,-179.065,6.181,148.838
C08014=1175.232,90.885,-51.146,-179.067,6.180,148.839
C08015=1175.237,90.636,-51.128,-179.070,6.179,148.839
C08016=1175.242,90.387,-51.111,-179.072,6.178,148.840
C08017=1175.247,90.137,-51.093,-179.075,6.176,148.840
C08018=1175.252,89.888,-51.075,-179.078,6.176,148.841
C08019=1175.257,89.639,-51.057,-179.081,6.174,148.841
C08020=1175.262,89.390,-51.039,-179.083,6.173,148.842
C08021=1175.267,89.141,-51.021,-179.086,6.172,148.843
C08022=1175.272,88.891,-51.005,-179.088,6.171,148.843
C08023=1175.276,88.642,-50.987,-179.091,6.169,148.843
C08024=1175.281,88.393,-50.969,-179.094,6.169,148.844
C08025=1175.286,88.144,-50.951,-179.096,6.167,148.844
C08026=1175.292,87.894,-50.933,-179.100,6.166,148.845
C08027=1175.296,87.645,-50.915,-179.102,6.165,148.845
C08028=1175.301,87.395,-50.898,-179.104,6.163,148.846
C08029=1175.307,87.146,-50.880,-179.107,6.163,148.847
C08030=1175.311,86.897,-50.863,-179.110,6.161,148.847
C08031=1175.316,86.648,-50.845,-179.112,6.160,148.848
C08032=1175.321,86.398,-50.828,-179.115,6.159,148.848
C08033=1175.326,86.149,-50.810,-179.118,6.158,148.849
C08034=1175.331,85.900,-50.792,-179.120,6.156,148.849
C08035=1175.336,85.650,-50.774,-179.123,6.156,148.850
C08036=1175.340,85.401,-50.757,-179.126,6.154,148.850
C08037=1175.345,85.152,-50.739,-179.128,6.153,148.851
C08038=1175.350,84.902,-50.722,-179.131,6.152,148.851
C08039=1175.355,84.653,-50.704,-179.133,6.151,148.852
C08040=1175.360,84.404,-50.686,-179.137,6.150,148.852
C08041=1175.365,84.154,-50.669,-179.139,6.149,148.853
C08042=1175.369,83.905,-50.651,-179.141,6.147,148.853
C08043=1175.375,83.655,-50.634,-179.144,6.147,148.854
C08044=1175.380,83.406,-50.616,-179.147,6.145,148.854
C08045=1175.384,83.156,-50.599,-179.149,6.144,148.855
C08046=1175.389,82.907,-50.581,-179.152,6.143,148.855
C08047=1175.394,82.657,-50.564,-179.155,6.142,148.856
C08048=1175.399,82.408,-50.546,-179.157,6.140,148.856
C08049=1175.404,82.159,-50.529,-179.160,6.140,148.857
C08050=1175.408,81.910,-50.511,-179.163,6.138,148.857
C08051=1175.414,81.660,-50.494,-179.165,6.137,148.858
C08052=1175.419,81.411,-50.476,-179.168,6.136,148.859
C08053=1175.424,81.162,-50.460,-179.170,6.135,148.859
C08054=1175.429,80.913,-50.442,-179.173,6.134,148.860
C08055=1175.434,80.644,-50.423,-179.176,6.133,148.860
C08056=1175.438,80.376,-50.404,-179.179,6.131,148.861
C08057=1175.444,80.108,-50.386,-179.182,6.130,148.861
C08058=1175.450,79.839,-50.367,-179.184,6.129,148.862
C08059=1175.455,79.590,-50.349,-179.187,6.128,148.862
C08060=1175.459,79.340,-50.333,-179.190,6.127,148.863
C08061=1175.464,79.090,-50.315,-179.193,6.126,148.864
C08062=1175.469,78.841,-50.297,-179.195,6.125,148.864
C08063=1175.474,78.592,-50.281,-179.198,6.123,148.865
C08064=1175.480,78.343,-50.264,-179.200,6.123,148.865
C08065=1175.484,78.094,-50.246,-179.203,6.121,148.865
C08066=1175.489,77.844,-50.229,-179.206,6.120,148.866
C08067=1175.494,77.594,-50.212,-179.208,6.119,148.867
C08068=1175.498,77.345,-50.195,-179.211,6.118,148.867
C08069=1175.504,77.095,-50.177,-179.213,6.117,148.868
C08070=1175.509,76.847,-50.161,-179.216,6.116,148.868
C08071=1175.514,76.598,-50.143,-179.218,6.115,148.869
C08072=1175.519,76.348,-50.126,-179.222,6.114,148.869
C08073=1175.523,76.098,-50.109,-179.224,6.113,148.870
C08074=1175.528,75.849,-50.091,-179.227,6.111,148.870
C08075=1175.533,75.600,-50.074,-179.229,6.110,148.871
C08076=1175.538,75.351,-50.058,-179.232,6.109,148.872
C08077=1175.543,75.101,-50.041,-179.235,6.108,148.872
C08078=1175.548,74.852,-50.023,-179.237,6.108,148.873
C08079=1175.552,74.602,-50.006,-179.240,6.106,148.873
C08080=1175.558,74.353,-49.989,-179.243,6.105,148.874
C08081=1175.563,74.104,-49.973,-179.245,6.104,148.874
C08082=1175.568,73.854,-49.955,-179.247,6.103,148.875
C08083=1175.572,73.605,-49.938,-179.251,6.102,148.875
C08084=1175.577,73.355,-49.921,-179.253,6.101,148.876
C08085=1175.582,73.107,-49.904,-179.255,6.100,148.876
C08086=1175.588,72.857,-49.887,-179.258,6.098,148.877
C08087=1175.592,72.607,-49.870,-179.261,6.098,148.877
C08088=1175.597,72.357,-49.853,-179.263,6.096,148.878
C08089=1175.602,72.109,-49.837,-179.266,6.096,148.878
C08090=1175.607,71.860,-49.819,-179.269,6.094,148.879
C08091=1175.612,71.610,-49.802,-179.271,6.093,148.880
C08092=1175.617,71.360,-49.785,-179.274,6.093,148.880
C08093=1175.622,71.111,-49.769,-179.277,6.091,148.881
C08094=1175.626,70.862,-49.752,-179.279,6.090,148.881
C08095=1175.632,70.612,-49.735,-179.282,6.089,148.882
C08096=1175.636,70.363,-49.718,-179.284,6.088,148.882
C08097=1175.642,70.114,-49.701,-179.287,6.088,148.883
C08098=1175.646,69.864,-49.685,-179.290,6.086,148.883
C08099=1175.651,69.615,-49.668,-179.292,6.085,148.884
C08100=1175.657,69.366,-49.651,-179.295,6.084,148.884
C08101=1175.661,69.116,-49.634,-179.298,6.083,148.885
C08102=1175.666,68.866,-49.617,-179.300,6.081,148.885
C08103=1175.671,68.617,-49.600,-179.303,6.081,148.886
C08104=1175.676,68.368,-49.584,-179.305,6.080,148.887
C08105=1175.681,68.118,-49.567,-179.308,6.079,148.887
C08106=1175.686,67.869,-49.550,-179.311,6.078,148.888
C08107=1175.691,67.620,-49.534,-179.314,6.077,148.888
C08108=1175.696,67.370,-49.517,-179.316,6.076,148.889
C08109=1175.700,67.121,-49.500,-179.319,6.075,148.889
C08110=1175.706,66.872,-49.484,-179.321,6.073,148.890
C08111=1175.711,66.622,-49.466,-179.324,6.073,148.890
C08112=1175.715,66.373,-49.450,-179.326,6.072,148.891
C08113=1175.720,66.124,-49.433,-179.329,6.071,148.892
C08114=1175.725,65.874,-49.417,-179.331,6.070,148.892
C08115=1175.730,65.624,-49.400,-179.335,6.068,148.893
C08116=1175.735,65.375,-49.384,-179.337,6.068,148.893
C08117=1175.740,65.126,-49.367,-179.339,6.067,148.894
C08118=1175.746,64.877,-49.350,-179.342,6.065,148.894
C08119=1175.750,64.627,-49.334,-179.345,6.065,148.895
C08120=1175.755,64.378,-49.317,-179.348,6.063,148.895
C08121=1175.760,64.128,-49.301,-179.350,6.063,148.896
C08122=1175.765,63.879,-49.285,-179.352,6.062,148.896
C08123=1175.770,63.629,-49.267,-179.356,6.060,148.897
C08124=1175.775,63.380,-49.251,-179.358,6.060,148.897
C08125=1175.779,63.131,-49.234,-179.360,6.059,148.898
C08126=1175.785,62.881,-49.219,-179.364,6.058,148.899
C08127=1175.790,62.631,-49.202,-179.366,6.057,148.899
C08128=1175.794,62.382,-49.185,-179.368,6.056,148.900
C08129=1175.800,62.133,-49.169,-179.371,6.055,148.900
C08130=1175.804,61.883,-49.153,-179.374,6.054,148.901
C08131=1175.809,61.634,-49.136,-179.376,6.052,148.901
C08132=1175.815,61.384,-49.119,-179.379,6.052,148.902
C08133=1175.820,61.135,-49.103,-179.381,6.051,148.903
C08134=1175.824,60.886,-49.087,-179.384,6.050,148.903
C08135=1175.829,60.636,-49.070,-179.387,6.049,148.904
C08136=1175.834,60.387,-49.054,-179.389,6.048,148.904
C08137=1175.839,60.137,-49.038,-179.392,6.047,148.905
C08138=1175.844,59.888,-49.022,-179.395,6.046,148.905
C08139=1175.849,59.639,-49.004,-179.397,6.045,148.906
C08140=1175.854,59.389,-48.989,-179.400,6.044,148.906
C08141=1175.859,59.140,-48.972,-179.402,6.043,148.907
C08142=1175.864,58.890,-48.956,-179.405,6.043,148.908
C08143=1175.869,58.641,-48.940,-179.408,6.041,148.908
C08144=1175.874,58.392,-48.924,-179.410,6.040,148.909
C08145=1175.879,58.142,-48.908,-179.413,6.040,148.909
C08146=1175.884,57.893,-48.891,-179.415,6.038,148.910
C08147=1175.889,57.643,-48.875,-179.418,6.038,148.910
C08148=1175.894,57.394,-48.858,-179.420,6.037,148.911
C08149=1175.899,57.145,-48.842,-179.423,6.035,148.912
C08150=1175.904,56.895,-48.826,-179.426,6.035,148.912
C08151=1175.909,56.646,-48.809,-179.428,6.034,148.913
C08152=1175.914,56.396,-48.794,-179.431,6.032,148.913
C08153=1175.919,56.147,-48.777,-179.434,6.032,148.914
C08154=1175.924,55.897,-48.762,-179.436,6.031,148.914
C08155=1175.928,55.648,-48.745,-179.439,6.030,148.915
C08156=1175.934,55.398,-48.729,-179.442,6.029,148.916
C08157=1175.938,55.149,-48.713,-179.444,6.028,148.916
C08158=1175.944,54.900,-48.697,-179.447,6.027,148.917
C08159=1175.949,54.631,-48.680,-179.449,6.026,148.917
C08160=1175.954,54.363,-48.662,-179.452,6.025,148.918
C08161=1175.959,54.094,-48.645,-179.455,6.024,148.918
C08162=1175.965,53.826,-48.628,-179.458,6.023,148.919
C08163=1175.970,53.575,-48.612,-179.460,6.022,148.919
C08164=1175.975,53.327,-48.596,-179.463,6.022,148.920
C08165=1175.980,53.077,-48.580,-179.466,6.020,148.921
C08166=1175.985,52.828,-48.563,-179.468,6.019,148.921
C08167=1175.990,52.578,-48.548,-179.471,6.018,148.922
C08168=1175.995,52.328,-48.532,-179.473,6.018,148.922
C08169=1176.000,52.080,-48.516,-179.476,6.017,148.923
C08170=1176.005,51.829,-48.500,-179.479,6.016,148.923
C08171=1176.010,51.581,-48.483,-179.481,6.015,148.924
C08172=1176.015,51.331,-48.468,-179.484,6.014,148.925
C08173=1176.019,51.081,-48.452,-179.487,6.013,148.925
C08174=1176.024,50.833,-48.436,-179.489,6.012,148.926
C08175=1176.029,50.583,-48.420,-179.491,6.012,148.926
C08176=1176.035,50.333,-48.405,-179.494,6.010,148.927
C08177=1176.040,50.084,-48.389,-179.497,6.009,148.927
C08178=1176.044,49.834,-48.372,-179.499,6.009,148.928
C08179=1176.050,49.585,-48.357,-179.502,6.007,148.929
C08180=1176.055,49.335,-48.341,-179.505,6.007,148.929
C08181=1176.059,49.086,-48.325,-179.507,6.006,148.930
C08182=1176.064,48.837,-48.309,-179.510,6.005,148.930
C08183=1176.070,48.587,-48.294,-179.512,6.004,148.931
C08184=1176.075,48.337,-48.278,-179.515,6.003,148.931
C08185=1176.080,48.089,-48.262,-179.518,6.003,148.932
C08186=1176.084,47.838,-48.246,-179.520,6.001,148.933
C08187=1176.090,47.589,-48.230,-179.523,6.001,148.933
C08188=1176.094,47.340,-48.215,-179.525,6.000,148.934
C08189=1176.099,47.090,-48.199,-179.528,5.999,148.934
C08190=1176.104,46.841,-48.183,-179.530,5.997,148.935
C08191=1176.110,46.592,-48.167,-179.533,5.997,148.935
C08192=1176.115,46.342,-48.152,-179.536,5.996,148.936
C08193=1176.119,46.093,-48.136,-179.538,5.996,148.937
C08194=1176.125,45.843,-48.121,-179.541,5.994,148.937
C08195=1176.130,45.594,-48.105,-179.543,5.993,148.938
C08196=1176.135,45.344,-48.089,-179.546,5.993,148.938
C08197=1176.139,45.095,-48.073,-179.548,5.992,148.939
C08198=1176.144,44.846,-48.058,-179.551,5.991,148.939
C08199=1176.149,44.596,-48.042,-179.554,5.990,148.940
C08200=1176.155,44.346,-48.026,-179.556,5.989,148.941
C08201=1176.159,44.097,-48.011,-179.559,5.988,148.941
C08202=1176.165,43.848,-47.996,-179.561,5.987,148.942
C08203=1176.169,43.598,-47.980,-179.564,5.987,148.942
C08204=1176.174,43.349,-47.965,-179.567,5.986,148.943
C08205=1176.179,43.099,-47.949,-179.569,5.985,148.944
C08206=1176.185,42.850,-47.934,-179.572,5.984,148.944
C08207=1176.190,42.600,-47.918,-179.574,5.983,148.945
C08208=1176.194,42.351,-47.903,-179.577,5.983,148.945
C08209=1176.200,42.101,-47.887,-179.579,5.982,148.946
C08210=1176.205,41.852,-47.871,-179.582,5.980,148.946
C08211=1176.209,41.602,-47.856,-179.585,5.980,148.947
C08212=1176.214,41.353,-47.841,-179.587,5.979,148.948
C08213=1176.220,41.103,-47.825,-179.590,5.979,148.948
C08214=1176.225,40.854,-47.810,-179.592,5.977,148.949
C08215=1176.229,40.604,-47.794,-179.595,5.976,148.949
C08216=1176.235,40.355,-47.778,-179.598,5.976,148.950
C08217=1176.239,40.105,-47.763,-179.600,5.975,148.950
C08218=1176.245,39.856,-47.748,-179.603,5.974,148.951
C08219=1176.250,39.607,-47.732,-179.605,5.973,148.952
C08220=1176.254,39.357,-47.717,-179.608,5.972,148.952
C08221=1176.260,39.107,-47.701,-179.611,5.972,148.953
C08222=1176.264,38.858,-47.686,-179.613,5.971,148.953
C08223=1176.270,38.609,-47.671,-179.616,5.970,148.954
C08224=1176.275,38.359,-47.656,-179.618,5.969,148.954
C08225=1176.279,38.109,-47.641,-179.621,5.968,148.955
C08226=1176.285,37.860,-47.625,-179.623,5.968,148.956
C08227=1176.289,37.611,-47.610,-179.626,5.966,148.956
C08228=1176.295,37.361,-47.594,-179.629,5.966,148.957
C08229=1176.299,37.112,-47.579,-179.631,5.965,148.957
C08230=1176.305,36.862,-47.564,-179.634,5.964,148.958
C08231=1176.310,36.613,-47.549,-179.636,5.964,148.959
C08232=1176.315,36.363,-47.534,-179.639,5.962,148.959
C08233=1176.320,36.114,-47.518,-179.642,5.962,148.960
C08234=1176.325,35.864,-47.503,-179.644,5.961,148.960
C08235=1176.330,35.614,-47.488,-179.646,5.960,148.961
C08236=1176.335,35.365,-47.473,-179.649,5.960,148.962
C08237=1176.340,35.116,-47.457,-179.652,5.958,148.962
C08238=1176.345,34.867,-47.442,-179.654,5.958,148.963
C08239=1176.350,34.616,-47.427,-179.657,5.957,148.963
C08240=1176.355,34.367,-47.412,-179.659,5.956,148.964
C08241=1176.360,34.118,-47.397,-179.662,5.956,148.965
C08242=1176.365,33.869,-47.382,-179.665,5.954,148.965
C08243=1176.370,33.618,-47.367,-179.667,5.954,148.966
C08244=1176.375,33.369,-47.352,-179.669,5.953,148.966
C08245=1176.380,33.120,-47.336,-179.672,5.952,148.967
C08246=1176.385,32.870,-47.322,-179.675,5.952,148.967
C08247=1176.390,32.621,-47.307,-179.677,5.951,148.968
C08248=1176.395,32.372,-47.291,-179.680,5.950,148.969
C08249=1176.400,32.121,-47.277,-179.683,5.949,148.969
C08250=1176.405,31.872,-47.261,-179.685,5.948,148.970
C08251=1176.410,31.623,-47.246,-179.688,5.948,148.970
C08252=1176.416,31.373,-47.231,-179.690,5.947,148.971
C08253=1176.420,31.124,-47.216,-179.693,5.946,148.972
C08254=1176.425,30.875,-47.201,-179.696,5.945,148.972
C08255=1176.431,30.625,-47.186,-179.698,5.944,148.973
C08256=1176.435,30.376,-47.171,-179.700,5.944,148.973
C08257=1176.441,30.126,-47.157,-179.703,5.943,148.974
C08258=1176.445,29.876,-47.142,-179.705,5.942,148.974
C08259=1176.450,29.627,-47.127,-179.708,5.941,148.975
C08260=1176.456,29.377,-47.112,-179.711,5.940,148.976
C08261=1176.460,29.128,-47.097,-179.713,5.940,148.976
C08262=1176.465,28.879,-47.082,-179.716,5.939,148.977
C08263=1176.471,28.609,-47.066,-179.718,5.938,148.977
C08264=1176.476,28.341,-47.050,-179.721,5.937,148.978
C08265=1176.482,28.072,-47.034,-179.724,5.937,148.979
C08266=1176.487,27.803,-47.018,-179.727,5.936,148.979
C08267=1176.492,27.554,-47.003,-179.730,5.935,148.980
C08268=1176.498,27.304,-46.989,-179.732,5.934,148.981
C08269=1176.502,27.055,-46.974,-179.735,5.934,148.981
C08270=1176.507,26.805,-46.959,-179.737,5.933,148.982
C08271=1176.513,26.555,-46.944,-179.739,5.932,148.982
C08272=1176.518,26.306,-46.929,-179.742,5.932,148.983
C08273=1176.522,26.057,-46.914,-179.744,5.931,148.984
C08274=1176.528,25.807,-46.900,-179.748,5.930,148.984
C08275=1176.533,25.558,-46.885,-179.750,5.929,148.985
C08276=1176.538,25.308,-46.870,-179.752,5.928,148.985
C08277=1176.543,25.058,-46.856,-179.755,5.928,148.986
C08278=1176.548,24.809,-46.840,-179.757,5.927,148.986
C08279=1176.553,24.559,-46.826,-179.760,5.926,148.987
C08280=1176.558,24.310,-46.811,-179.762,5.926,148.988
C08281=1176.563,24.060,-46.797,-179.765,5.924,148.988
C08282=1176.568,23.810,-46.782,-179.768,5.924,148.989
C08283=1176.573,23.561,-46.767,-179.770,5.923,148.990
C08284=1176.578,23.311,-46.753,-179.773,5.922,148.990
C08285=1176.583,23.062,-46.738,-179.775,5.922,148.991
C08286=1176.588,22.813,-46.724,-179.777,5.921,148.991
C08287=1176.594,22.563,-46.709,-179.780,5.921,148.992
C08288=1176.599,22.314,-46.695,-179.783,5.920,148.993
C08289=1176.603,22.064,-46.680,-179.785,5.918,148.993
C08290=1176.608,21.815,-46.665,-179.788,5.918,148.994
C08291=1176.613,21.565,-46.651,-179.791,5.917,148.994
C08292=1176.618,21.315,-46.637,-179.793,5.917,148.995
C08293=1176.624,21.066,-46.621,-179.796,5.916,148.996
C08294=1176.629,20.816,-46.607,-179.798,5.916,148.996
C08295=1176.634,20.566,-46.593,-179.800,5.915,148.997
C08296=1176.638,20.317,-46.578,-179.803,5.914,148.997
C08297=1176.644,20.068,-46.564,-179.805,5.913,148.998
C08298=1176.649,19.819,-46.550,-179.808,5.912,148.998
C08299=1176.654,19.569,-46.535,-179.811,5.912,148.999
C08300=1176.659,19.319,-46.520,-179.813,5.911,149.000
C08301=1176.664,19.070,-46.505,-179.816,5.910,149.000
C08302=1176.669,18.820,-46.491,-179.819,5.910,149.001
C08303=1176.674,18.570,-46.477,-179.821,5.909,149.001
C08304=1176.679,18.321,-46.463,-179.823,5.909,149.002
C08305=1176.684,18.072,-46.449,-179.826,5.908,149.003
C08306=1176.689,17.822,-46.434,-179.828,5.907,149.003
C08307=1176.694,17.573,-46.419,-179.831,5.906,149.004
C08308=1176.699,17.323,-46.405,-179.834,5.905,149.005
C08309=1176.704,17.073,-46.391,-179.836,5.905,149.005
C08310=1176.709,16.824,-46.377,-179.839,5.904,149.006
C08311=1176.715,16.574,-46.362,-179.841,5.903,149.006
C08312=1176.720,16.325,-46.348,-179.844,5.903,149.007
C08313=1176.725,16.075,-46.333,-179.846,5.902,149.008
C08314=1176.730,15.825,-46.319,-179.849,5.901,149.008
C08315=1176.735,15.576,-46.304,-179.851,5.901,149.009
C08316=1176.740,15.327,-46.290,-179.854,5.900,149.009
C08317=1176.745,15.078,-46.276,-179.856,5.900,149.010
C08318=1176.750,14.828,-46.262,-179.859,5.899,149.011
C08319=1176.755,14.578,-46.247,-179.862,5.898,149.011
C08320=1176.760,14.328,-46.233,-179.864,5.897,149.012
C08321=1176.766,14.079,-46.219,-179.867,5.897,149.012
C08322=1176.771,13.830,-46.205,-179.869,5.896,149.013
C08323=1176.776,13.580,-46.191,-179.872,5.895,149.013
C08324=1176.780,13.330,-46.176,-179.874,5.895,149.014
C08325=1176.785,13.081,-46.162,-179.877,5.894,149.015
C08326=1176.791,12.832,-46.148,-179.879,5.893,149.015
C08327=1176.796,12.582,-46.134,-179.882,5.893,149.016
C08328=1176.801,12.332,-46.120,-179.884,5.892,149.016
C08329=1176.806,12.082,-46.105,-179.886,5.892,149.017
C08330=1176.811,11.834,-46.092,-179.889,5.891,149.018
C08331=1176.816,11.584,-46.078,-179.891,5.890,149.018
C08332=1176.821,11.334,-46.064,-179.894,5.889,149.019
C08333=1176.826,11.085,-46.049,-179.897,5.889,149.020
C08334=1176.831,10.835,-46.036,-179.899,5.888,149.020
C08335=1176.836,10.585,-46.022,-179.902,5.887,149.021
C08336=1176.841,10.336,-46.008,-179.905,5.887,149.021
C08337=1176.846,10.086,-45.993,-179.907,5.886,149.022
C08338=1176.852,9.837,-45.979,-179.909,5.885,149.023
C08339=1176.857,9.587,-45.965,-179.912,5.885,149.023
C08340=1176.862,9.337,-45.951,-179.914,5.884,149.024
C08341=1176.867,9.089,-45.937,-179.917,5.884,149.024
C08342=1176.872,8.838,-45.924,-179.920,5.883,149.025
C08343=1176.877,8.589,-45.910,-179.922,5.882,149.026
C08344=1176.882,8.339,-45.895,-179.924,5.882,149.026
C08345=1176.887,8.090,-45.881,-179.927,5.881,149.027
C08346=1176.892,7.840,-45.867,-179.929,5.880,149.027
C08347=1176.897,7.590,-45.853,-179.932,5.880,149.028
C08348=1176.902,7.341,-45.840,-179.934,5.880,149.029
C08349=1176.907,7.091,-45.826,-179.937,5.879,149.029
C08350=1176.912,6.842,-45.812,-179.939,5.878,149.030
C08351=1176.918,6.593,-45.798,-179.942,5.878,149.031
C08352=1176.923,6.343,-45.784,-179.944,5.877,149.031
C08353=1176.927,6.093,-45.771,-179.947,5.876,149.032
C08354=1176.933,5.844,-45.757,-179.950,5.875,149.032
C08355=1176.938,5.594,-45.742,-179.952,5.874,149.033
C08356=1176.943,5.345,-45.728,-179.955,5.874,149.034
C08357=1176.949,5.095,-45.715,-179.958,5.873,149.034
C08358=1176.953,4.846,-45.701,-179.960,5.873,149.035
C08359=1176.958,4.596,-45.687,-179.962,5.872,149.035
C08360=1176.964,4.346,-45.674,-179.965,5.872,149.036
C08361=1176.969,4.097,-45.659,-179.967,5.871,149.037
C08362=1176.973,3.848,-45.646,-179.970,5.870,149.037
C08363=1176.979,3.597,-45.633,-179.972,5.869,149.038
C08364=1176.984,3.348,-45.618,-179.975,5.869,149.038
C08365=1176.989,3.099,-45.604,-179.977,5.869,149.039
C08366=1176.994,2.849,-45.591,-179.979,5.868,149.040
C08367=1176.999,2.579,-45.576,-179.982,5.867,149.040
C08368=1177.005,2.311,-45.562,-179.985,5.867,149.041
C08369=1177.011,2.041,-45.547,-179.987,5.866,149.042
C08370=1177.016,1.772,-45.532,-179.991,5.865,149.042
C08371=1177.021,1.522,-45.518,-179.993,5.865,149.043
C08372=1177.026,1.273,-45.505,-179.995,5.864,149.043
C08373=1177.031,1.023,-45.491,-179.998,5.863,149.044
C08374=1177.037,0.774,-45.477,179.999,5.863,149.045
C08375=1177.041,0.524,-45.464,179.997,5.862,149.045
C08376=1177.046,0.274,-45.450,179.994,5.861,149.046
C08377=1177.052,0.025,-45.436,179.992,5.861,149.047
C08378=1177.056,-0.225,-45.423,179.990,5.860,149.047
C08379=1177.062,-0.474,-45.409,179.987,5.860,149.048
C08380=1177.067,-0.724,-45.395,179.984,5.859,149.049
C08381=1177.072,-0.973,-45.383,179.982,5.858,149.049
C08382=1177.077,-1.223,-45.368,179.979,5.858,149.050
C08383=1177.083,-1.473,-45.355,179.977,5.857,149.050
C08384=1177.087,-1.722,-45.341,179.975,5.857,149.051
C08385=1177.093,-1.972,-45.328,179.972,5.856,149.052
C08386=1177.097,-2.221,-45.315,179.969,5.856,149.052
C08387=1177.102,-2.471,-45.301,179.967,5.855,149.053
C08388=1177.108,-2.720,-45.287,179.964,5.854,149.053
C08389=1177.113,-2.971,-45.274,179.962,5.855,149.054
C08390=1177.118,-3.220,-45.260,179.960,5.854,149.055
C08391=1177.123,-3.470,-45.247,179.958,5.853,149.055
C08392=1177.128,-3.719,-45.233,179.955,5.853,149.056
C08393=1177.133,-3.969,-45.220,179.953,5.852,149.056
C08394=1177.139,-4.218,-45.207,179.950,5.852,149.057
C08395=1177.144,-4.468,-45.193,179.947,5.851,149.058
C08396=1177.149,-4.717,-45.180,179.945,5.850,149.058
C08397=1177.154,-4.967,-45.166,179.943,5.850,149.059
C08398=1177.159,-5.216,-45.153,179.940,5.849,149.060
C08399=1177.164,-5.467,-45.140,179.938,5.849,149.060
C08400=1177.169,-5.715,-45.127,179.935,5.848,149.061
C08401=1177.174,-5.966,-45.113,179.932,5.848,149.061
C08402=1177.179,-6.214,-45.100,179.930,5.847,149.062
C08403=1177.185,-6.464,-45.086,179.928,5.846,149.063
C08404=1177.189,-6.714,-45.073,179.925,5.846,149.063
C08405=1177.195,-6.963,-45.060,179.923,5.845,149.064
C08406=1177.199,-7.213,-45.047,179.920,5.845,149.064
C08407=1177.205,-7.463,-45.033,179.918,5.844,149.065
C08408=1177.210,-7.713,-45.020,179.915,5.843,149.066
C08409=1177.215,-7.962,-45.007,179.913,5.843,149.066
C08410=1177.220,-8.212,-44.994,179.910,5.842,149.067
C08411=1177.226,-8.461,-44.980,179.908,5.842,149.067
C08412=1177.230,-8.711,-44.967,179.905,5.841,149.068
C08413=1177.236,-8.960,-44.953,179.903,5.841,149.069
C08414=1177.241,-9.210,-44.941,179.900,5.840,149.069
C08415=1177.245,-9.460,-44.928,179.898,5.839,149.070
C08416=1177.251,-9.709,-44.914,179.895,5.839,149.071
C08417=1177.255,-9.959,-44.901,179.893,5.838,149.071
C08418=1177.261,-10.208,-44.888,179.890,5.838,149.072
C08419=1177.266,-10.458,-44.875,179.888,5.838,149.073
C08420=1177.271,-10.707,-44.861,179.886,5.837,149.073
C08421=1177.277,-10.957,-44.848,179.883,5.837,149.074
C08422=1177.281,-11.207,-44.835,179.881,5.836,149.074
C08423=1177.287,-11.456,-44.822,179.878,5.835,149.075
C08424=1177.291,-11.706,-44.809,179.876,5.835,149.076
C08425=1177.297,-11.956,-44.796,179.873,5.834,149.076
C08426=1177.302,-12.205,-44.783,179.871,5.834,149.077
C08427=1177.307,-12.455,-44.770,179.868,5.833,149.077
C08428=1177.312,-12.704,-44.757,179.866,5.833,149.078
C08429=1177.318,-12.954,-44.744,179.863,5.832,149.079
C08430=1177.322,-13.204,-44.731,179.861,5.831,149.079
C08431=1177.328,-13.453,-44.718,179.858,5.831,149.080
C08432=1177.333,-13.703,-44.705,179.856,5.830,149.081
C08433=1177.338,-13.953,-44.692,179.853,5.830,149.081
C08434=1177.343,-14.202,-44.678,179.851,5.829,149.082
C08435=1177.348,-14.452,-44.665,179.849,5.830,149.082
C08436=1177.353,-14.701,-44.653,179.846,5.829,149.083
C08437=1177.359,-14.951,-44.640,179.844,5.828,149.084
C08438=1177.363,-15.201,-44.627,179.841,5.828,149.084
C08439=1177.368,-15.450,-44.614,179.839,5.827,149.085
C08440=1177.374,-15.700,-44.601,179.836,5.827,149.085
C08441=1177.379,-15.950,-44.588,179.834,5.826,149.086
C08442=1177.384,-16.199,-44.575,179.831,5.825,149.087
C08443=1177.390,-16.448,-44.562,179.829,5.825,149.087
C08444=1177.394,-16.699,-44.549,179.826,5.824,149.088
C08445=1177.399,-16.948,-44.536,179.824,5.824,149.088
C08446=1177.404,-17.197,-44.524,179.821,5.823,149.089
C08447=1177.410,-17.447,-44.511,179.819,5.823,149.090
C08448=1177.415,-17.697,-44.498,179.817,5.823,149.090
C08449=1177.420,-17.946,-44.485,179.814,5.822,149.091
C08450=1177.425,-18.195,-44.473,179.812,5.822,149.092
C08451=1177.430,-18.446,-44.459,179.810,5.821,149.092
C08452=1177.436,-18.695,-44.446,179.807,5.820,149.093
C08453=1177.441,-18.944,-44.434,179.804,5.820,149.094
C08454=1177.446,-19.194,-44.421,179.802,5.819,149.094
C08455=1177.451,-19.444,-44.408,179.799,5.819,149.095
C08456=1177.456,-19.693,-44.395,179.797,5.818,149.095
C08457=1177.461,-19.943,-44.382,179.795,5.817,149.096
C08458=1177.467,-20.193,-44.370,179.793,5.818,149.097
C08459=1177.471,-20.443,-44.358,179.790,5.817,149.097
C08460=1177.477,-20.692,-44.344,179.788,5.816,149.098
C08461=1177.482,-20.942,-44.332,179.785,5.816,149.098
C08462=1177.487,-21.191,-44.319,179.782,5.816,149.099
C08463=1177.492,-21.441,-44.306,179.780,5.815,149.100
C08464=1177.497,-21.690,-44.294,179.778,5.814,149.100
C08465=1177.502,-21.940,-44.281,179.775,5.814,149.101
C08466=1177.508,-22.190,-44.268,179.773,5.813,149.101
C08467=1177.513,-22.440,-44.256,179.771,5.813,149.102
C08468=1177.518,-22.689,-44.243,179.768,5.813,149.103
C08469=1177.523,-22.938,-44.230,179.766,5.812,149.103
C08470=1177.528,-23.188,-44.218,179.763,5.812,149.104
C08471=1177.534,-23.458,-44.204,179.760,5.811,149.105
C08472=1177.539,-23.728,-44.190,179.758,5.811,149.105
C08473=1177.545,-23.997,-44.177,179.755,5.810,149.106
C08474=1177.551,-24.267,-44.163,179.752,5.810,149.107
C08475=1177.556,-24.517,-44.151,179.750,5.809,149.107
C08476=1177.561,-24.766,-44.138,179.748,5.809,149.108
C08477=1177.566,-25.016,-44.126,179.745,5.808,149.109
C08478=1177.571,-25.266,-44.113,179.743,5.807,149.109
C08479=1177.576,-25.516,-44.101,179.740,5.807,149.110
C08480=1177.581,-25.765,-44.088,179.738,5.807,149.111
C08481=1177.586,-26.014,-44.076,179.736,5.806,149.111
C08482=1177.592,-26.264,-44.063,179.733,5.806,149.112
C08483=1177.596,-26.514,-44.051,179.731,5.806,149.112
C08484=1177.602,-26.764,-44.038,179.728,5.805,149.113
C08485=1177.607,-27.013,-44.026,179.726,5.804,149.114
C08486=1177.612,-27.263,-44.014,179.723,5.804,149.114
C08487=1177.618,-27.513,-44.001,179.721,5.803,149.115
C08488=1177.623,-27.762,-43.988,179.719,5.803,149.115
C08489=1177.628,-28.012,-43.976,179.716,5.803,149.116
C08490=1177.633,-28.262,-43.963,179.714,5.802,149.117
C08491=1177.638,-28.511,-43.951,179.711,5.802,149.117
C08492=1177.644,-28.761,-43.939,179.709,5.801,149.118
C08493=1177.649,-29.010,-43.926,179.706,5.801,149.119
C08494=1177.654,-29.260,-43.913,179.704,5.800,149.119
C08495=1177.659,-29.510,-43.902,179.702,5.800,149.120
C08496=1177.664,-29.759,-43.889,179.699,5.800,149.121
C08497=1177.669,-30.010,-43.877,179.697,5.799,149.121
C08498=1177.674,-30.259,-43.864,179.694,5.799,149.122
C08499=1177.679,-30.508,-43.852,179.692,5.798,149.122
C08500=1177.684,-30.758,-43.840,179.689,5.797,149.123
C08501=1177.689,-31.007,-43.828,179.687,5.798,149.124
C08502=1177.695,-31.257,-43.816,179.685,5.797,149.124
C08503=1177.700,-31.506,-43.803,179.682,5.796,149.125
C08504=1177.705,-31.756,-43.791,179.680,5.796,149.125
C08505=1177.710,-32.006,-43.779,179.677,5.796,149.126
C08506=1177.716,-32.256,-43.767,179.675,5.795,149.127
C08507=1177.721,-32.505,-43.754,179.672,5.794,149.127
C08508=1177.726,-32.756,-43.742,179.670,5.795,149.128
C08509=1177.731,-33.005,-43.729,179.668,5.794,149.129
C08510=1177.736,-33.255,-43.717,179.665,5.793,149.129
C08511=1177.741,-33.504,-43.705,179.663,5.793,149.130
C08512=1177.747,-33.754,-43.693,179.661,5.792,149.130
C08513=1177.751,-34.003,-43.681,179.658,5.792,149.131
C08514=1177.757,-34.253,-43.669,179.656,5.792,149.132
C08515=1177.762,-34.502,-43.656,179.654,5.791,149.132
C08516=1177.767,-34.752,-43.645,179.651,5.791,149.133
C08517=1177.772,-35.002,-43.632,179.648,5.790,149.134
C08518=1177.778,-35.252,-43.620,179.646,5.790,149.134
C08519=1177.783,-35.501,-43.607,179.643,5.789,149.135
C08520=1177.788,-35.751,-43.596,179.641,5.789,149.136
C08521=1177.793,-36.000,-43.584,179.639,5.789,149.136
C08522=1177.798,-36.250,-43.572,179.637,5.788,149.137
C08523=1177.804,-36.500,-43.560,179.634,5.788,149.137
C08524=1177.809,-36.749,-43.547,179.632,5.787,149.138
C08525=1177.814,-36.999,-43.535,179.630,5.787,149.139
C08526=1177.820,-37.249,-43.523,179.627,5.787,149.139
C08527=1177.824,-37.498,-43.511,179.625,5.786,149.140
C08528=1177.829,-37.748,-43.500,179.622,5.786,149.140
C08529=1177.835,-37.998,-43.488,179.619,5.785,149.141
C08530=1177.840,-38.247,-43.475,179.617,5.784,149.142
C08531=1177.845,-38.497,-43.463,179.615,5.785,149.142
C08532=1177.850,-38.747,-43.452,179.613,5.784,149.143
C08533=1177.855,-38.996,-43.439,179.610,5.783,149.143
C08534=1177.861,-39.246,-43.427,179.608,5.783,149.144
C08535=1177.866,-39.496,-43.416,179.605,5.783,149.145
C08536=1177.871,-39.745,-43.403,179.603,5.783,149.145
C08537=1177.876,-39.995,-43.392,179.601,5.782,149.146
C08538=1177.881,-40.245,-43.380,179.598,5.782,149.147
C08539=1177.887,-40.495,-43.368,179.596,5.781,149.147
C08540=1177.892,-40.744,-43.355,179.593,5.780,149.148
C08541=1177.896,-40.994,-43.344,179.591,5.781,149.149
C08542=1177.902,-41.244,-43.332,179.589,5.780,149.149
C08543=1177.907,-41.493,-43.320,179.586,5.780,149.150
C08544=1177.912,-41.743,-43.308,179.584,5.779,149.151
C08545=1177.917,-41.992,-43.296,179.582,5.778,149.151
C08546=1177.923,-42.242,-43.284,179.579,5.779,149.152
C08547=1177.929,-42.492,-43.273,179.577,5.778,149.152
C08548=1177.933,-42.741,-43.261,179.575,5.777,149.153
C08549=1177.938,-42.990,-43.249,179.572,5.777,149.154
C08550=1177.944,-43.240,-43.237,179.570,5.777,149.154
C08551=1177.949,-43.490,-43.226,179.568,5.777,149.155
C08552=1177.954,-43.740,-43.214,179.565,5.776,149.155
C08553=1177.959,-43.990,-43.202,179.562,5.776,149.156
C08554=1177.964,-44.239,-43.190,179.560,5.775,149.157
C08555=1177.969,-44.489,-43.178,179.558,5.775,149.157
C08556=1177.975,-44.739,-43.166,179.555,5.775,149.158
C08557=1177.979,-44.988,-43.155,179.553,5.774,149.158
C08558=1177.985,-45.238,-43.144,179.551,5.774,149.159
C08559=1177.991,-45.488,-43.132,179.548,5.773,149.160
C08560=1177.996,-45.737,-43.120,179.546,5.773,149.160
C08561=1178.001,-45.987,-43.108,179.544,5.773,149.161
C08562=1178.006,-46.236,-43.096,179.541,5.772,149.162
C08563=1178.011,-46.486,-43.085,179.539,5.771,149.162
C08564=1178.016,-46.736,-43.073,179.537,5.772,149.163
C08565=1178.022,-46.986,-43.061,179.535,5.771,149.163
C08566=1178.027,-47.235,-43.050,179.532,5.771,149.164
C08567=1178.032,-47.485,-43.038,179.529,5.770,149.165
C08568=1178.037,-47.734,-43.027,179.528,5.770,149.165
C08569=1178.042,-47.984,-43.015,179.525,5.770,149.166
C08570=1178.048,-48.234,-43.003,179.522,5.769,149.167
C08571=1178.053,-48.484,-42.992,179.520,5.768,149.167
C08572=1178.058,-48.734,-42.980,179.517,5.768,149.168
C08573=1178.063,-48.983,-42.969,179.515,5.768,149.169
C08574=1178.069,-49.233,-42.957,179.513,5.768,149.169
C08575=1178.074,-49.503,-42.944,179.511,5.767,149.170
C08576=1178.080,-49.773,-42.932,179.508,5.767,149.170
C08577=1178.086,-50.044,-42.919,179.505,5.766,149.171
C08578=1178.091,-50.314,-42.906,179.503,5.766,149.172
C08579=1178.096,-50.564,-42.895,179.501,5.766,149.172
C08580=1178.102,-50.813,-42.883,179.498,5.765,149.173
C08581=1178.107,-51.063,-42.873,179.496,5.765,149.174
C08582=1178.112,-51.313,-42.861,179.493,5.764,149.174
C08583=1178.117,-51.563,-42.850,179.491,5.765,149.175
C08584=1178.122,-51.813,-42.838,179.489,5.764,149.176
C08585=1178.127,-52.062,-42.827,179.486,5.763,149.176
C08586=1178.133,-52.312,-42.815,179.484,5.763,149.177
C08587=1178.138,-52.561,-42.804,179.482,5.763,149.178
C08588=1178.143,-52.811,-42.792,179.480,5.763,149.178
C08589=1178.148,-53.060,-42.781,179.477,5.762,149.179
C08590=1178.154,-53.310,-42.769,179.474,5.762,149.179
C08591=1178.158,-53.560,-42.758,179.473,5.762,149.180
C08592=1178.164,-53.810,-42.746,179.470,5.761,149.181
C08593=1178.169,-54.060,-42.735,179.467,5.761,149.181
C08594=1178.175,-54.309,-42.724,179.465,5.760,149.182
C08595=1178.180,-54.559,-42.712,179.463,5.760,149.182
C08596=1178.184,-54.808,-42.701,179.461,5.760,149.183
C08597=1178.190,-55.058,-42.689,179.458,5.759,149.184
C08598=1178.195,-55.307,-42.678,179.456,5.759,149.184
C08599=1178.201,-55.558,-42.667,179.454,5.759,149.185
C08600=1178.205,-55.807,-42.656,179.451,5.758,149.186
C08601=1178.210,-56.057,-42.644,179.449,5.758,149.186
C08602=1178.216,-56.306,-42.633,179.446,5.757,149.187
C08603=1178.221,-56.556,-42.622,179.444,5.757,149.187
C08604=1178.227,-56.806,-42.611,179.442,5.757,149.188
C08605=1178.231,-57.056,-42.599,179.439,5.756,149.189
C08606=1178.237,-57.305,-42.588,179.437,5.757,149.189
C08607=1178.242,-57.555,-42.576,179.435,5.756,149.190
C08608=1178.247,-57.804,-42.565,179.433,5.755,149.190
C08609=1178.253,-58.054,-42.554,179.430,5.755,149.191
C08610=1178.258,-58.304,-42.543,179.428,5.755,149.192
C08611=1178.262,-58.554,-42.532,179.426,5.755,149.192
C08612=1178.268,-58.804,-42.520,179.423,5.754,149.193
C08613=1178.273,-59.053,-42.510,179.421,5.753,149.194
C08614=1178.278,-59.303,-42.498,179.419,5.754,149.194
C08615=1178.284,-59.553,-42.486,179.416,5.753,149.195
C08616=1178.289,-59.802,-42.476,179.414,5.752,149.195
C08617=1178.294,-60.052,-42.465,179.412,5.753,149.196
C08618=1178.299,-60.302,-42.453,179.409,5.752,149.197
C08619=1178.305,-60.551,-42.443,179.407,5.752,149.197
C08620=1178.310,-60.801,-42.432,179.404,5.751,149.198
C08621=1178.315,-61.051,-42.420,179.403,5.751,149.199
C08622=1178.321,-61.300,-42.409,179.400,5.751,149.199
C08623=1178.325,-61.550,-42.398,179.397,5.750,149.200
C08624=1178.330,-61.800,-42.387,179.396,5.750,149.200
C08625=1178.336,-62.049,-42.376,179.393,5.750,149.201
C08626=1178.341,-62.299,-42.365,179.390,5.750,149.202
C08627=1178.346,-62.549,-42.354,179.389,5.750,149.202
C08628=1178.352,-62.799,-42.343,179.386,5.749,149.203
C08629=1178.357,-63.048,-42.331,179.383,5.749,149.204
C08630=1178.362,-63.298,-42.321,179.381,5.748,149.204
C08631=1178.367,-63.547,-42.310,179.379,5.748,149.205
C08632=1178.372,-63.797,-42.298,179.377,5.747,149.205
C08633=1178.377,-64.048,-42.287,179.374,5.747,149.206
C08634=1178.383,-64.297,-42.277,179.372,5.747,149.207
C08635=1178.388,-64.547,-42.266,179.370,5.747,149.207
C08636=1178.394,-64.796,-42.254,179.367,5.746,149.208
C08637=1178.399,-65.046,-42.244,179.365,5.747,149.209
C08638=1178.403,-65.296,-42.233,179.363,5.746,149.209
C08639=1178.409,-65.545,-42.222,179.360,5.745,149.210
C08640=1178.414,-65.795,-42.211,179.358,5.745,149.210
C08641=1178.420,-66.044,-42.200,179.356,5.745,149.211
C08642=1178.425,-66.295,-42.189,179.354,5.745,149.212
C08643=1178.429,-66.544,-42.178,179.351,5.744,149.212
C08644=1178.435,-66.794,-42.168,179.349,5.744,149.213
C08645=1178.440,-67.044,-42.156,179.347,5.744,149.214
C08646=1178.446,-67.293,-42.145,179.344,5.743,149.214
C08647=1178.451,-67.543,-42.134,179.342,5.743,149.215
C08648=1178.456,-67.792,-42.124,179.340,5.743,149.215
C08649=1178.461,-68.043,-42.113,179.337,5.742,149.216
C08650=1178.466,-68.292,-42.102,179.335,5.742,149.217
C08651=1178.472,-68.542,-42.091,179.333,5.742,149.217
C08652=1178.477,-68.792,-42.080,179.331,5.741,149.218
C08653=1178.483,-69.041,-42.070,179.329,5.741,149.218
C08654=1178.487,-69.291,-42.058,179.326,5.741,149.219
C08655=1178.493,-69.540,-42.048,179.324,5.740,149.220
C08656=1178.498,-69.791,-42.038,179.322,5.740,149.220
C08657=1178.503,-70.040,-42.027,179.319,5.740,149.221
C08658=1178.509,-70.290,-42.016,179.317,5.740,149.222
C08659=1178.514,-70.540,-42.004,179.315,5.740,149.222
C08660=1178.519,-70.789,-41.994,179.312,5.739,149.223
C08661=1178.524,-71.040,-41.984,179.310,5.738,149.223
C08662=1178.530,-71.288,-41.973,179.308,5.739,149.224
C08663=1178.535,-71.539,-41.962,179.305,5.738,149.225
C08664=1178.540,-71.788,-41.952,179.303,5.738,149.225
C08665=1178.545,-72.038,-41.941,179.301,5.738,149.226
C08666=1178.550,-72.287,-41.930,179.299,5.737,149.226
C08667=1178.555,-72.537,-41.919,179.296,5.737,149.227
C08668=1178.561,-72.787,-41.908,179.294,5.737,149.228
C08669=1178.566,-73.037,-41.898,179.292,5.736,149.228
C08670=1178.572,-73.287,-41.887,179.289,5.736,149.229
C08671=1178.577,-73.536,-41.876,179.288,5.736,149.230
C08672=1178.582,-73.786,-41.866,179.285,5.736,149.230
C08673=1178.587,-74.036,-41.855,179.282,5.735,149.231
C08674=1178.593,-74.285,-41.844,179.281,5.735,149.231
C08675=1178.598,-74.535,-41.834,179.278,5.735,149.232
C08676=1178.603,-74.785,-41.824,179.276,5.734,149.233
C08677=1178.609,-75.034,-41.813,179.274,5.734,149.233
C08678=1178.614,-75.284,-41.802,179.271,5.734,149.234
C08679=1178.619,-75.556,-41.791,179.269,5.733,149.234
C08680=1178.625,-75.826,-41.780,179.266,5.733,149.235
C08681=1178.631,-76.097,-41.768,179.264,5.733,149.236
C08682=1178.637,-76.369,-41.756,179.262,5.733,149.237
C08683=1178.642,-76.618,-41.746,179.259,5.732,149.237
C08684=1178.648,-76.867,-41.735,179.257,5.732,149.238
C08685=1178.653,-77.117,-41.725,179.255,5.732,149.239
C08686=1178.658,-77.367,-41.714,179.253,5.731,149.239
C08687=1178.663,-77.617,-41.704,179.250,5.731,149.240
C08688=1178.668,-77.866,-41.694,179.248,5.731,149.240
C08689=1178.673,-78.116,-41.683,179.246,5.730,149.241
C08690=1178.678,-78.366,-41.673,179.244,5.731,149.242
C08691=1178.684,-78.615,-41.662,179.241,5.730,149.242
C08692=1178.689,-78.865,-41.652,179.239,5.729,149.243
C08693=1178.695,-79.115,-41.642,179.237,5.729,149.243
C08694=1178.700,-79.365,-41.631,179.234,5.729,149.244
C08695=1178.705,-79.615,-41.621,179.232,5.729,149.245
C08696=1178.710,-79.864,-41.610,179.230,5.729,149.245
C08697=1178.716,-80.114,-41.599,179.227,5.728,149.246
C08698=1178.721,-80.363,-41.589,179.226,5.728,149.246
C08699=1178.726,-80.614,-41.579,179.223,5.728,149.247
C08700=1178.732,-80.863,-41.568,179.221,5.727,149.248
C08701=1178.737,-81.113,-41.558,179.219,5.727,149.248
C08702=1178.742,-81.363,-41.548,179.216,5.727,149.249
C08703=1178.747,-81.612,-41.538,179.214,5.726,149.249
C08704=1178.752,-81.863,-41.527,179.212,5.727,149.250
C08705=1178.758,-82.112,-41.517,179.210,5.726,149.251
C08706=1178.763,-82.361,-41.506,179.208,5.726,149.251
C08707=1178.768,-82.611,-41.496,179.205,5.726,149.252
C08708=1178.774,-82.861,-41.485,179.203,5.725,149.253
C08709=1178.779,-83.110,-41.475,179.201,5.725,149.253
C08710=1178.784,-83.361,-41.465,179.199,5.725,149.254
C08711=1178.789,-83.610,-41.455,179.196,5.724,149.254
C08712=1178.794,-83.860,-41.445,179.194,5.724,149.255
C08713=1178.800,-84.110,-41.434,179.192,5.724,149.256
C08714=1178.805,-84.359,-41.424,179.190,5.724,149.256
C08715=1178.810,-84.609,-41.414,179.187,5.723,149.257
C08716=1178.816,-84.859,-41.403,179.185,5.723,149.258
C08717=1178.821,-85.108,-41.394,179.183,5.723,149.258
C08718=1178.826,-85.358,-41.383,179.180,5.723,149.259
C08719=1178.831,-85.608,-41.373,179.178,5.722,149.259
C08720=1178.837,-85.857,-41.363,179.176,5.722,149.260
C08721=1178.842,-86.108,-41.352,179.173,5.722,149.261
C08722=1178.847,-86.357,-41.343,179.172,5.722,149.261
C08723=1178.853,-86.607,-41.333,179.169,5.722,149.262
C08724=1178.858,-86.857,-41.322,179.167,5.721,149.262
C08725=1178.863,-87.107,-41.312,179.165,5.721,149.263
C08726=1178.868,-87.356,-41.303,179.163,5.720,149.264
C08727=1178.873,-87.606,-41.292,179.161,5.721,149.264
C08728=1178.879,-87.856,-41.282,179.158,5.720,149.265
C08729=1178.884,-88.105,-41.272,179.156,5.720,149.265
C08730=1178.890,-88.355,-41.261,179.154,5.720,149.266
C08731=1178.894,-88.605,-41.251,179.152,5.719,149.267
C08732=1178.900,-88.854,-41.241,179.149,5.720,149.267
C08733=1178.905,-89.104,-41.231,179.147,5.719,149.268
C08734=1178.910,-89.355,-41.222,179.145,5.718,149.269
C08735=1178.916,-89.604,-41.212,179.143,5.718,149.269
C08736=1178.921,-89.854,-41.201,179.140,5.718,149.270
C08737=1178.927,-90.103,-41.191,179.138,5.718,149.270
C08738=1178.931,-90.353,-41.181,179.136,5.718,149.271
C08739=1178.937,-90.603,-41.171,179.133,5.717,149.272
C08740=1178.943,-90.853,-41.161,179.132,5.717,149.272
C08741=1178.948,-91.102,-41.151,179.129,5.717,149.273
C08742=1178.952,-91.352,-41.141,179.128,5.717,149.273
C08743=1178.958,-91.602,-41.131,179.125,5.716,149.274
C08744=1178.964,-91.851,-41.121,179.123,5.716,149.274
C08745=1178.969,-92.101,-41.112,179.121,5.716,149.275
C08746=1178.974,-92.352,-41.101,179.118,5.715,149.276
C08747=1178.979,-92.601,-41.091,179.116,5.716,149.276
C08748=1178.984,-92.850,-41.082,179.114,5.715,149.277
C08749=1178.990,-93.100,-41.071,179.111,5.714,149.278
C08750=1178.995,-93.351,-41.062,179.109,5.715,149.278
C08751=1179.000,-93.600,-41.052,179.107,5.714,149.279
C08752=1179.006,-93.849,-41.042,179.105,5.714,149.279
C08753=1179.011,-94.099,-41.031,179.103,5.714,149.280
C08754=1179.016,-94.349,-41.023,179.101,5.714,149.281
C08755=1179.021,-94.599,-41.012,179.099,5.713,149.281
C08756=1179.027,-94.849,-41.002,179.096,5.713,149.282
C08757=1179.032,-95.099,-40.993,179.094,5.713,149.282
C08758=1179.038,-95.348,-40.983,179.092,5.713,149.283
C08759=1179.043,-95.597,-40.973,179.090,5.713,149.284
C08760=1179.048,-95.848,-40.963,179.087,5.712,149.284
C08761=1179.053,-96.098,-40.953,179.085,5.713,149.285
C08762=1179.058,-96.347,-40.943,179.083,5.712,149.285
C08763=1179.064,-96.596,-40.933,179.080,5.711,149.286
C08764=1179.069,-96.846,-40.924,179.079,5.711,149.287
C08765=1179.074,-97.097,-40.914,179.076,5.711,149.287
C08766=1179.080,-97.347,-40.904,179.075,5.711,149.288
C08767=1179.085,-97.596,-40.895,179.072,5.711,149.289
C08768=1179.090,-97.846,-40.884,179.070,5.711,149.289
C08769=1179.096,-98.095,-40.875,179.068,5.710,149.290
C08770=1179.101,-98.345,-40.865,179.065,5.709,149.290
C08771=1179.105,-98.595,-40.855,179.063,5.710,149.291
C08772=1179.111,-98.845,-40.846,179.061,5.709,149.291
C08773=1179.117,-99.095,-40.836,179.059,5.709,149.292
C08774=1179.122,-99.344,-40.827,179.057,5.709,149.293
C08775=1179.128,-99.594,-40.816,179.055,5.709,149.293
C08776=1179.133,-99.843,-40.807,179.053,5.708,149.294
C08777=1179.138,-100.093,-40.797,179.050,5.708,149.295
C08778=1179.143,-100.343,-40.787,179.048,5.708,149.295
C08779=1179.149,-100.593,-40.778,179.046,5.708,149.296
C08780=1179.154,-100.843,-40.768,179.044,5.708,149.296
C08781=1179.159,-101.093,-40.759,179.041,5.707,149.297
C08782=1179.164,-101.342,-40.749,179.039,5.708,149.298
C08783=1179.171,-101.614,-40.738,179.037,5.707,149.298
C08784=1179.176,-101.886,-40.728,179.034,5.706,149.299
C08785=1179.182,-102.157,-40.718,179.032,5.707,149.300
C08786=1179.187,-102.429,-40.707,179.030,5.706,149.300
C08787=1179.193,-102.679,-40.698,179.027,5.706,149.301
C08788=1179.198,-102.928,-40.688,179.026,5.706,149.301
C08789=1179.204,-103.178,-40.679,179.023,5.705,149.302
C08790=1179.208,-103.428,-40.669,179.022,5.705,149.302
C08791=1179.214,-103.678,-40.659,179.019,5.705,149.303
C08792=1179.219,-103.928,-40.650,179.017,5.705,149.304
C08793=1179.225,-104.178,-40.640,179.015,5.705,149.304
C08794=1179.230,-104.427,-40.631,179.012,5.704,149.305
C08795=1179.235,-104.677,-40.622,179.010,5.704,149.306
C08796=1179.241,-104.926,-40.611,179.008,5.703,149.306
C08797=1179.246,-105.176,-40.603,179.006,5.704,149.307
C08798=1179.252,-105.426,-40.593,179.004,5.703,149.307
C08799=1179.256,-105.676,-40.583,179.002,5.703,149.308
C08800=1179.262,-105.926,-40.574,179.000,5.703,149.308
C08801=1179.267,-106.175,-40.564,178.998,5.703,149.309
C08802=1179.272,-106.425,-40.555,178.995,5.702,149.310
C08803=1179.277,-106.675,-40.545,178.993,5.703,149.310
C08804=1179.283,-106.925,-40.536,178.991,5.702,149.311
C08805=1179.288,-107.175,-40.526,178.989,5.702,149.312
C08806=1179.293,-107.424,-40.517,178.987,5.702,149.312
C08807=1179.298,-107.674,-40.508,178.984,5.701,149.313
C08808=1179.304,-107.924,-40.498,178.983,5.701,149.313
C08809=1179.309,-108.174,-40.489,178.980,5.701,149.314
C08810=1179.314,-108.423,-40.480,178.978,5.701,149.314
C08811=1179.320,-108.673,-40.470,178.976,5.700,149.315
C08812=1179.325,-108.923,-40.461,178.974,5.700,149.316
C08813=1179.331,-109.173,-40.451,178.971,5.700,149.316
C08814=1179.336,-109.422,-40.442,178.970,5.700,149.317
C08815=1179.341,-109.672,-40.433,178.967,5.700,149.318
C08816=1179.347,-109.922,-40.423,178.965,5.700,149.318
C08817=1179.352,-110.172,-40.414,178.963,5.699,149.319
C08818=1179.357,-110.421,-40.405,178.961,5.699,149.319
C08819=1179.363,-110.672,-40.395,178.958,5.699,149.320
C08820=1179.368,-110.921,-40.386,178.957,5.699,149.320
C08821=1179.373,-111.171,-40.377,178.954,5.699,149.321
C08822=1179.379,-111.421,-40.367,178.952,5.698,149.322
C08823=1179.384,-111.671,-40.358,178.950,5.698,149.322
C08824=1179.389,-111.920,-40.350,178.948,5.697,149.323
C08825=1179.394,-112.170,-40.340,178.946,5.697,149.323
C08826=1179.400,-112.420,-40.330,178.943,5.697,149.324
C08827=1179.405,-112.670,-40.322,178.942,5.697,149.325
C08828=1179.410,-112.920,-40.313,178.939,5.697,149.325
C08829=1179.416,-113.169,-40.302,178.938,5.697,149.326
C08830=1179.421,-113.419,-40.294,178.935,5.696,149.326
C08831=1179.426,-113.669,-40.285,178.933,5.696,149.327
C08832=1179.431,-113.919,-40.276,178.931,5.696,149.328
C08833=1179.437,-114.168,-40.266,178.929,5.696,149.328
C08834=1179.443,-114.417,-40.257,178.926,5.696,149.329
C08835=1179.448,-114.667,-40.248,178.925,5.696,149.329
C08836=1179.453,-114.917,-40.239,178.923,5.695,149.330
C08837=1179.459,-115.167,-40.230,178.921,5.695,149.331
C08838=1179.464,-115.417,-40.221,178.918,5.695,149.331
C08839=1179.469,-115.666,-40.211,178.916,5.695,149.332
C08840=1179.474,-115.916,-40.202,178.914,5.694,149.332
C08841=1179.480,-116.166,-40.193,178.912,5.695,149.333
C08842=1179.485,-116.416,-40.184,178.910,5.694,149.333
C08843=1179.490,-116.666,-40.175,178.908,5.694,149.334
C08844=1179.496,-116.916,-40.166,178.905,5.693,149.335
C08845=1179.502,-117.166,-40.157,178.903,5.694,149.335
C08846=1179.506,-117.415,-40.147,178.901,5.693,149.336
C08847=1179.512,-117.665,-40.138,178.900,5.693,149.336
C08848=1179.517,-117.914,-40.130,178.897,5.693,149.337
C08849=1179.522,-118.164,-40.121,178.895,5.693,149.337
C08850=1179.528,-118.414,-40.112,178.893,5.692,149.338
C08851=1179.534,-118.664,-40.102,178.891,5.692,149.339
C08852=1179.539,-118.914,-40.093,178.888,5.692,149.339
C08853=1179.544,-119.164,-40.084,178.887,5.692,149.340
C08854=1179.549,-119.414,-40.076,178.885,5.691,149.340
C08855=1179.554,-119.664,-40.067,178.882,5.692,149.341
C08856=1179.559,-119.913,-40.058,178.880,5.691,149.342
C08857=1179.566,-120.163,-40.049,178.878,5.691,149.342
C08858=1179.571,-120.412,-40.039,178.876,5.691,149.343
C08859=1179.576,-120.662,-40.030,178.874,5.691,149.344
C08860=1179.581,-120.912,-40.021,178.872,5.690,149.344
C08861=1179.586,-121.162,-40.012,178.870,5.690,149.344
C08862=1179.591,-121.411,-40.003,178.867,5.690,149.345
C08863=1179.597,-121.661,-39.995,178.866,5.690,149.346
C08864=1179.602,-121.911,-39.986,178.863,5.689,149.346
C08865=1179.608,-122.161,-39.977,178.862,5.689,149.347
C08866=1179.613,-122.411,-39.968,178.859,5.689,149.348
C08867=1179.619,-122.660,-39.959,178.857,5.689,149.348
C08868=1179.624,-122.910,-39.950,178.855,5.688,149.349
C08869=1179.629,-123.160,-39.941,178.853,5.689,149.349
C08870=1179.634,-123.410,-39.932,178.851,5.688,149.350
C08871=1179.640,-123.659,-39.924,178.849,5.688,149.350
C08872=1179.645,-123.909,-39.915,178.847,5.688,149.351
C08873=1179.650,-124.159,-39.906,178.845,5.688,149.351
C08874=1179.656,-124.409,-39.898,178.842,5.687,149.352
C08875=1179.661,-124.659,-39.889,178.841,5.687,149.353
C08876=1179.667,-124.909,-39.879,178.838,5.687,149.353
C08877=1179.672,-125.158,-39.871,178.836,5.687,149.354
C08878=1179.678,-125.408,-39.862,178.834,5.686,149.354
C08879=1179.683,-125.658,-39.853,178.832,5.687,149.355
C08880=1179.688,-125.908,-39.844,178.830,5.686,149.356
C08881=1179.693,-126.158,-39.835,178.828,5.686,149.356
C08882=1179.699,-126.407,-39.827,178.826,5.686,149.357
C08883=1179.704,-126.657,-39.818,178.824,5.686,149.357
C08884=1179.710,-126.907,-39.809,178.821,5.685,149.358
C08885=1179.715,-127.157,-39.801,178.820,5.685,149.358
C08886=1179.720,-127.407,-39.792,178.818,5.686,149.359
C08887=1179.299,-127.418,-39.832,178.814,5.689,149.361
C08888=1179.294,-127.168,-39.841,178.816,5.688,149.360
C08889=1179.288,-126.919,-39.849,178.818,5.689,149.360
C08890=1179.282,-126.668,-39.858,178.820,5.689,149.359
C08891=1179.277,-126.418,-39.867,178.822,5.690,149.359
C08892=1179.272,-126.168,-39.875,178.824,5.690,149.358
C08893=1179.267,-125.919,-39.884,178.827,5.690,149.357
C08894=1179.261,-125.669,-39.893,178.828,5.690,149.357
C08895=1179.256,-125.420,-39.902,178.830,5.691,149.356
C08896=1179.251,-125.170,-39.911,178.832,5.690,149.356
C08897=1179.246,-124.920,-39.920,178.835,5.691,149.355
C08898=1179.240,-124.670,-39.928,178.837,5.691,149.355
C08899=1179.235,-124.420,-39.937,178.839,5.691,149.354
C08900=1179.229,-124.171,-39.946,178.841,5.691,149.354
C08901=1179.223,-123.920,-39.955,178.843,5.691,149.353
C08902=1179.218,-123.670,-39.964,178.845,5.692,149.352
C08903=1179.213,-123.420,-39.972,178.847,5.691,149.352
C08904=1179.208,-123.171,-39.981,178.849,5.692,149.351
C08905=1179.203,-122.921,-39.990,178.851,5.692,149.350
C08906=1179.197,-122.672,-39.999,178.853,5.692,149.350
C08907=1179.192,-122.422,-40.008,178.855,5.692,149.349
C08908=1179.187,-122.172,-40.017,178.858,5.693,149.349
C08909=1179.181,-121.922,-40.026,178.859,5.693,149.348
C08910=1179.176,-121.672,-40.034,178.862,5.693,149.348
C08911=1179.170,-121.422,-40.044,178.864,5.693,149.347
C08912=1179.165,-121.173,-40.052,178.866,5.694,149.347
C08913=1179.159,-120.923,-40.061,178.868,5.693,149.346
C08914=1179.154,-120.673,-40.070,178.870,5.694,149.345
C08915=1179.149,-120.423,-40.079,178.872,5.694,149.345
C08916=1179.144,-120.174,-40.088,178.874,5.695,149.344
C08917=1179.139,-119.924,-40.097,178.876,5.694,149.343
C08918=1179.134,-119.674,-40.106,178.879,5.695,149.343
C08919=1179.128,-119.424,-40.116,178.880,5.695,149.342
C08920=1179.122,-119.175,-40.125,178.883,5.695,149.342
C08921=1179.117,-118.925,-40.133,178.884,5.695,149.341
C08922=1179.112,-118.675,-40.142,178.887,5.696,149.341
C08923=1179.107,-118.426,-40.151,178.889,5.696,149.340
C08924=1179.101,-118.176,-40.160,178.891,5.696,149.339
C08925=1179.096,-117.926,-40.170,178.893,5.696,149.339
C08926=1179.090,-117.676,-40.179,178.895,5.697,149.338
C08927=1179.085,-117.426,-40.187,178.897,5.696,149.338
C08928=1179.080,-117.176,-40.196,178.899,5.697,149.337
C08929=1179.075,-116.926,-40.205,178.902,5.697,149.336
C08930=1179.069,-116.677,-40.215,178.904,5.697,149.336
C08931=1179.064,-116.427,-40.224,178.906,5.697,149.335
C08932=1179.058,-116.178,-40.233,178.908,5.698,149.335
C08933=1179.053,-115.928,-40.242,178.910,5.698,149.334
C08934=1179.048,-115.678,-40.251,178.912,5.698,149.334
C08935=1179.042,-115.428,-40.260,178.914,5.698,149.333
C08936=1179.037,-115.179,-40.270,178.917,5.698,149.332
C08937=1179.032,-114.929,-40.279,178.918,5.698,149.332
C08938=1179.027,-114.679,-40.288,178.921,5.699,149.331
C08939=1179.021,-114.429,-40.297,178.922,5.699,149.331
C08940=1179.016,-114.179,-40.306,178.925,5.699,149.330
C08941=1179.011,-113.929,-40.315,178.927,5.700,149.329
C08942=1179.006,-113.680,-40.324,178.929,5.700,149.329
C08943=1179.000,-113.430,-40.334,178.932,5.700,149.328
C08944=1178.995,-113.180,-40.343,178.933,5.700,149.328
C08945=1178.990,-112.930,-40.352,178.936,5.701,149.327
C08946=1178.984,-112.680,-40.362,178.937,5.701,149.327
C08947=1178.979,-112.430,-40.371,178.940,5.701,149.326
C08948=1178.974,-112.181,-40.380,178.942,5.701,149.325
C08949=1178.969,-111.931,-40.389,178.944,5.701,149.325
C08950=1178.962,-111.682,-40.399,178.946,5.701,149.324
C08951=1178.957,-111.432,-40.407,178.949,5.702,149.323
C08952=1178.952,-111.182,-40.416,178.950,5.702,149.323
C08953=1178.946,-110.932,-40.426,178.953,5.702,149.322
C08954=1178.941,-110.683,-40.435,178.955,5.702,149.322
C08955=1178.936,-110.433,-40.444,178.957,5.703,149.321
C08956=1178.930,-110.183,-40.454,178.959,5.703,149.321
C08957=1178.925,-109.934,-40.463,178.961,5.703,149.320
C08958=1178.920,-109.684,-40.472,178.963,5.703,149.319
C08959=1178.914,-109.434,-40.482,178.965,5.704,149.319
C08960=1178.909,-109.184,-40.491,178.967,5.703,149.318
C08961=1178.904,-108.934,-40.500,178.970,5.704,149.318
C08962=1178.898,-108.684,-40.510,178.972,5.704,149.317
C08963=1178.894,-108.434,-40.519,178.974,5.704,149.317
C08964=1178.889,-108.185,-40.529,178.977,5.705,149.316
C08965=1178.883,-107.934,-40.538,178.978,5.705,149.315
C08966=1178.878,-107.685,-40.548,178.981,5.705,149.315
C08967=1178.872,-107.435,-40.557,178.982,5.705,149.314
C08968=1178.867,-107.185,-40.566,178.985,5.706,149.313
C08969=1178.862,-106.936,-40.576,178.987,5.705,149.313
C08970=1178.856,-106.686,-40.585,178.989,5.706,149.312
C08971=1178.851,-106.436,-40.594,178.991,5.706,149.312
C08972=1178.845,-106.186,-40.604,178.994,5.706,149.311
C08973=1178.840,-105.936,-40.613,178.995,5.706,149.311
C08974=1178.835,-105.687,-40.623,178.998,5.707,149.310
C08975=1178.830,-105.437,-40.632,179.000,5.707,149.309
C08976=1178.825,-105.188,-40.642,179.002,5.707,149.309
C08977=1178.819,-104.938,-40.652,179.004,5.708,149.308
C08978=1178.814,-104.688,-40.660,179.006,5.707,149.307
C08979=1178.808,-104.438,-40.671,179.009,5.708,149.307
C08980=1178.803,-104.188,-40.680,179.011,5.708,149.306
C08981=1178.799,-103.938,-40.689,179.013,5.709,149.306
C08982=1178.793,-103.688,-40.699,179.015,5.708,149.305
C08983=1178.788,-103.439,-40.709,179.017,5.709,149.305
C08984=1178.782,-103.189,-40.718,179.019,5.708,149.304
C08985=1178.777,-102.940,-40.728,179.022,5.709,149.303
C08986=1178.771,-102.690,-40.737,179.024,5.710,149.303
C08987=1178.766,-102.440,-40.747,179.026,5.710,149.302
C08988=1178.761,-102.168,-40.757,179.028,5.710,149.301
C08989=1178.755,-101.896,-40.768,179.031,5.710,149.301
C08990=1178.748,-101.625,-40.778,179.033,5.710,149.300
C08991=1178.743,-101.354,-40.789,179.035,5.711,149.299
C08992=1178.737,-101.103,-40.798,179.037,5.710,149.299
C08993=1178.733,-100.854,-40.808,179.040,5.711,149.298
C08994=1178.727,-100.603,-40.818,179.042,5.712,149.298
C08995=1178.722,-100.354,-40.827,179.044,5.712,149.297
C08996=1178.716,-100.104,-40.837,179.047,5.712,149.296
C08997=1178.712,-99.855,-40.846,179.048,5.712,149.296
C08998=1178.706,-99.605,-40.856,179.051,5.712,149.295
C08999=1178.701,-99.355,-40.865,179.053,5.712,149.295
C09000=1178.695,-99.106,-40.876,179.055,5.713,149.294
C09001=1178.691,-98.855,-40.885,179.057,5.713,149.294
C09002=1178.685,-98.606,-40.895,179.059,5.713,149.293
C09003=1178.680,-98.356,-40.904,179.062,5.714,149.292
C09004=1178.674,-98.106,-40.914,179.064,5.713,149.292
C09005=1178.669,-97.857,-40.924,179.066,5.714,149.291
C09006=1178.664,-97.607,-40.933,179.068,5.714,149.290
C09007=1178.658,-97.357,-40.944,179.070,5.715,149.290
C09008=1178.654,-97.107,-40.954,179.073,5.715,149.289
C09009=1178.648,-96.857,-40.963,179.074,5.715,149.289
C09010=1178.642,-96.608,-40.973,179.077,5.715,149.288
C09011=1178.637,-96.359,-40.983,179.079,5.715,149.288
C09012=1178.631,-96.108,-40.992,179.081,5.716,149.287
C09013=1178.627,-95.858,-41.002,179.083,5.716,149.286
C09014=1178.622,-95.609,-41.013,179.086,5.716,149.286
C09015=1178.616,-95.359,-41.022,179.088,5.717,149.285
C09016=1178.611,-95.109,-41.032,179.090,5.716,149.284
C09017=1178.605,-94.860,-41.042,179.093,5.717,149.284
C09018=1178.600,-94.610,-41.051,179.094,5.717,149.283
C09019=1178.595,-94.360,-41.061,179.097,5.717,149.283
C09020=1178.589,-94.110,-41.072,179.098,5.717,149.282
C09021=1178.585,-93.861,-41.081,179.101,5.718,149.281
C09022=1178.579,-93.611,-41.091,179.103,5.718,149.281
C09023=1178.574,-93.361,-41.101,179.105,5.718,149.280
C09024=1178.569,-93.111,-41.111,179.108,5.719,149.280
C09025=1178.563,-92.861,-41.120,179.110,5.718,149.279
C09026=1178.557,-92.612,-41.131,179.112,5.719,149.278
C09027=1178.552,-92.363,-41.140,179.115,5.720,149.278
C09028=1178.547,-92.112,-41.151,179.116,5.720,149.277
C09029=1178.542,-91.863,-41.161,179.119,5.720,149.277
C09030=1178.537,-91.613,-41.170,179.121,5.720,149.276
C09031=1178.531,-91.363,-41.180,179.123,5.720,149.275
C09032=1178.526,-91.113,-41.191,179.125,5.720,149.275
C09033=1178.521,-90.864,-41.200,179.127,5.721,149.274
C09034=1178.516,-90.614,-41.210,179.130,5.721,149.273
C09035=1178.510,-90.364,-41.220,179.132,5.721,149.273
C09036=1178.505,-90.114,-41.230,179.134,5.722,149.272
C09037=1178.500,-89.865,-41.240,179.136,5.722,149.272
C09038=1178.494,-89.615,-41.250,179.139,5.722,149.271
C09039=1178.489,-89.365,-41.261,179.141,5.723,149.271
C09040=1178.484,-89.115,-41.271,179.143,5.722,149.270
C09041=1178.479,-88.866,-41.281,179.146,5.723,149.269
C09042=1178.473,-88.616,-41.290,179.147,5.723,149.269
C09043=1178.468,-88.366,-41.301,179.150,5.723,149.268
C09044=1178.463,-88.116,-41.310,179.152,5.724,149.267
C09045=1178.457,-87.867,-41.321,179.154,5.723,149.267
C09046=1178.452,-87.617,-41.331,179.156,5.724,149.266
C09047=1178.447,-87.367,-41.341,179.159,5.725,149.266
C09048=1178.441,-87.118,-41.352,179.161,5.725,149.265
C09049=1178.436,-86.868,-41.361,179.163,5.725,149.264
C09050=1178.431,-86.618,-41.372,179.165,5.725,149.264
C09051=1178.426,-86.369,-41.382,179.167,5.725,149.263
C09052=1178.420,-86.119,-41.392,179.170,5.726,149.262
C09053=1178.416,-85.869,-41.402,179.172,5.726,149.262
C09054=1178.410,-85.619,-41.412,179.174,5.726,149.261
C09055=1178.404,-85.369,-41.422,179.176,5.726,149.261
C09056=1178.399,-85.119,-41.432,179.179,5.727,149.260
C09057=1178.394,-84.870,-41.443,179.181,5.727,149.259
C09058=1178.388,-84.620,-41.453,179.183,5.727,149.259
C09059=1178.384,-84.370,-41.463,179.186,5.727,149.258
C09060=1178.378,-84.121,-41.473,179.187,5.727,149.258
C09061=1178.373,-83.871,-41.483,179.190,5.728,149.257
C09062=1178.368,-83.621,-41.494,179.192,5.729,149.257
C09063=1178.362,-83.371,-41.504,179.194,5.728,149.256
C09064=1178.357,-83.121,-41.515,179.197,5.729,149.255
C09065=1178.352,-82.872,-41.524,179.199,5.729,149.255
C09066=1178.347,-82.622,-41.534,179.201,5.729,149.254
C09067=1178.342,-82.373,-41.546,179.203,5.730,149.253
C09068=1178.336,-82.123,-41.556,179.205,5.729,149.253
C09069=1178.331,-81.874,-41.566,179.208,5.730,149.252
C09070=1178.326,-81.623,-41.577,179.210,5.731,149.252
C09071=1178.320,-81.374,-41.587,179.212,5.730,149.251
C09072=1178.315,-81.123,-41.598,179.215,5.731,149.250
C09073=1178.310,-80.874,-41.607,179.217,5.731,149.250
C09074=1178.305,-80.625,-41.617,179.219,5.731,149.249
C09075=1178.300,-80.374,-41.628,179.221,5.732,149.248
C09076=1178.294,-80.125,-41.638,179.224,5.733,149.248
C09077=1178.289,-79.875,-41.648,179.226,5.732,149.247
C09078=1178.284,-79.625,-41.659,179.228,5.733,149.247
C09079=1178.278,-79.376,-41.670,179.230,5.733,149.246
C09080=1178.273,-79.126,-41.680,179.233,5.733,149.245
C09081=1178.268,-78.876,-41.691,179.235,5.734,149.245
C09082=1178.263,-78.626,-41.701,179.237,5.733,149.244
C09083=1178.257,-78.377,-41.711,179.240,5.734,149.243
C09084=1178.252,-78.127,-41.722,179.242,5.735,149.243
C09085=1178.247,-77.877,-41.733,179.244,5.734,149.242
C09086=1178.241,-77.628,-41.743,179.246,5.735,149.242
C09087=1178.236,-77.378,-41.754,179.249,5.735,149.241
C09088=1178.231,-77.128,-41.764,179.250,5.735,149.241
C09089=1178.226,-76.878,-41.774,179.253,5.736,149.240
C09090=1178.220,-76.628,-41.785,179.255,5.735,149.239
C09091=1178.215,-76.379,-41.796,179.257,5.736,149.239
C09092=1178.210,-76.108,-41.807,179.260,5.737,149.238
C09093=1178.204,-75.837,-41.818,179.263,5.737,149.237
C09094=1178.198,-75.567,-41.829,179.265,5.737,149.237
C09095=1178.192,-75.295,-41.841,179.267,5.737,149.236
C09096=1178.187,-75.045,-41.851,179.270,5.738,149.235
C09097=1178.182,-74.796,-41.862,179.272,5.738,149.235
C09098=1178.176,-74.546,-41.873,179.274,5.738,149.234
C09099=1178.171,-74.296,-41.883,179.277,5.739,149.233
C09100=1178.166,-74.047,-41.894,179.279,5.739,149.233
C09101=1178.161,-73.797,-41.905,179.281,5.739,149.232
C09102=1178.155,-73.547,-41.915,179.283,5.739,149.232
C09103=1178.150,-73.297,-41.925,179.286,5.740,149.231
C09104=1178.145,-73.048,-41.936,179.288,5.740,149.230
C09105=1178.140,-72.798,-41.947,179.290,5.741,149.230
C09106=1178.134,-72.548,-41.958,179.293,5.741,149.229
C09107=1178.129,-72.298,-41.969,179.295,5.741,149.229
C09108=1178.124,-72.049,-41.979,179.297,5.742,149.228
C09109=1178.119,-71.799,-41.990,179.300,5.742,149.227
C09110=1178.113,-71.550,-42.001,179.302,5.742,149.227
C09111=1178.108,-71.299,-42.011,179.304,5.742,149.226
C09112=1178.103,-71.050,-42.022,179.306,5.743,149.225
C09113=1178.098,-70.800,-42.033,179.308,5.743,149.225
C09114=1178.092,-70.551,-42.043,179.311,5.743,149.224
C09115=1178.088,-70.301,-42.054,179.313,5.744,149.224
C09116=1178.081,-70.051,-42.065,179.315,5.744,149.223
C09117=1178.076,-69.801,-42.076,179.318,5.744,149.222
C09118=1178.072,-69.551,-42.087,179.320,5.745,149.222
C09119=1178.066,-69.302,-42.097,179.322,5.744,149.221
C09120=1178.061,-69.052,-42.108,179.325,5.745,149.220
C09121=1178.056,-68.803,-42.119,179.327,5.746,149.220
C09122=1178.051,-68.552,-42.129,179.329,5.745,149.219
C09123=1178.045,-68.303,-42.141,179.331,5.746,149.219
C09124=1178.040,-68.053,-42.151,179.334,5.746,149.218
C09125=1178.034,-67.804,-42.162,179.336,5.746,149.217
C09126=1178.029,-67.554,-42.173,179.338,5.747,149.217
C09127=1178.025,-67.304,-42.184,179.341,5.747,149.216
C09128=1178.019,-67.055,-42.194,179.343,5.747,149.215
C09129=1178.014,-66.805,-42.206,179.345,5.748,149.215
C09130=1178.008,-66.555,-42.216,179.348,5.748,149.214
C09131=1178.003,-66.305,-42.228,179.349,5.748,149.214
C09132=1177.998,-66.056,-42.238,179.352,5.749,149.213
C09133=1177.993,-65.806,-42.249,179.354,5.749,149.212
C09134=1177.987,-65.556,-42.260,179.357,5.750,149.212
C09135=1177.982,-65.307,-42.271,179.359,5.749,149.211
C09136=1177.977,-65.057,-42.282,179.361,5.750,149.211
C09137=1177.972,-64.808,-42.293,179.364,5.751,149.210
C09138=1177.966,-64.557,-42.304,179.366,5.750,149.209
C09139=1177.961,-64.307,-42.315,179.368,5.751,149.209
C09140=1177.956,-64.058,-42.326,179.371,5.751,149.208
C09141=1177.951,-63.808,-42.337,179.373,5.751,149.207
C09142=1177.946,-63.559,-42.348,179.375,5.752,149.207
C09143=1177.940,-63.309,-42.359,179.377,5.752,149.206
C09144=1177.935,-63.059,-42.370,179.380,5.753,149.206
C09145=1177.930,-62.810,-42.380,179.382,5.753,149.205
C09146=1177.924,-62.560,-42.392,179.384,5.753,149.204
C09147=1177.920,-62.310,-42.404,179.387,5.754,149.204
C09148=1177.914,-62.061,-42.414,179.389,5.753,149.203
